	            #tempMoveBlkVariantRetVal := MOVE_BLK_VARIANT(SRC := #In_EventStatus.sts_Events,
	                                                                 COUNT := INT_TO_UDINT(#In_EventStatus.sts_NumEvents),
	                                                                 SRC_INDEX := 0,
	                                                                 DEST_INDEX := 0,
	                                                                 DEST => #Sts_EventSummation.sts_Events);
	            #Sts_EventSummation.sts_NumEvents := #In_EventStatus.sts_NumEvents;
	        ELSE
	            
	            #tempMoveBlkVariantRetVal := MOVE_BLK_VARIANT(SRC := #In_EventStatus.sts_Events,
	                                                                 COUNT := INT_TO_UDINT (#Sts_EventSummation.wrk_EventArraySize),
	                                                                 SRC_INDEX := 0,
	                                                                 DEST_INDEX := 0,
	                                                                 DEST => #Sts_EventSummation.sts_Events);
	            #Sts_EventSummation.sts_NumEvents := #Sts_EventSummation.wrk_EventArraySize;
	            #Sts_ErrorCode := 1;
	        END_IF;
	    
	   
	    END_IF;    
	END_IF;
	
	// update the output
	#Sts_NumEvents := #Sts_EventSummation.sts_NumEvents;
	
	// Set Category Bits
	#Sts_EventSummation.wrk_Category_0_Latched := (#Sts_EventSummation.wrk_Category_0_Latched OR #In_EventStatus.sts_Category_0_Latched);
	#Sts_EventSummation.wrk_Category_1_Latched := (#Sts_EventSummation.wrk_Category_1_Latched OR #In_EventStatus.sts_Category_1_Latched);
	#Sts_EventSummation.wrk_Category_2_Latched := (#Sts_EventSummation.wrk_Category_2_Latched OR #In_EventStatus.sts_Category_2_Latched);
	#Sts_EventSummation.wrk_Category_3_Latched := (#Sts_EventSummation.wrk_Category_3_Latched OR #In_EventStatus.sts_Category_3_Latched);
	#Sts_EventSummation.wrk_Category_4_Latched := (#Sts_EventSummation.wrk_Category_4_Latched OR #In_EventStatus.sts_Category_4_Latched);
	#Sts_EventSummation.wrk_Category_5_Latched := (#Sts_EventSummation.wrk_Category_5_Latched OR #In_EventStatus.sts_Category_5_Latched);
	#Sts_EventSummation.wrk_Category_6_Latched := (#Sts_EventSummation.wrk_Category_6_Latched OR #In_EventStatus.sts_Category_6_Latched);
	#Sts_EventSummation.wrk_Category_7_Latched := (#Sts_EventSummation.wrk_Category_7_Latched OR #In_EventStatus.sts_Category_7_Latched);
	#Sts_EventSummation.wrk_Category_8_Latched := (#Sts_EventSummation.wrk_Category_8_Latched OR #In_EventStatus.sts_Category_8_Latched);
	#Sts_EventSummation.wrk_Category_9_Latched := (#Sts_EventSummation.wrk_Category_9_Latched OR #In_EventStatus.sts_Category_9_Latched);
	
	#Sts_Category_0_Latched := #In_EventStatus.sts_Category_0_Latched;
	#Sts_Category_1_Latched := #In_EventStatus.sts_Category_1_Latched;
	#Sts_Category_2_Latched := #In_EventStatus.sts_Category_2_Latched;
	#Sts_Category_3_Latched := #In_EventStatus.sts_Category_3_Latched;
	#Sts_Category_4_Latched := #In_EventStatus.sts_Category_4_Latched;
	#Sts_Category_5_Latched := #In_EventStatus.sts_Category_5_Latched;
	#Sts_Category_6_Latched := #In_EventStatus.sts_Category_6_Latched;
	#Sts_Category_7_Latched := #In_EventStatus.sts_Category_7_Latched;
	#Sts_Category_8_Latched := #In_EventStatus.sts_Category_8_Latched;
	#Sts_Category_9_Latched := #In_EventStatus.sts_Category_9_Latched;
	
	#Sts_EventSummation.wrk_Category_0_NotLatched := #Sts_EventSummation.wrk_Category_0_NotLatched OR #In_EventStatus.sts_Category_0_NotLatched;
	#Sts_EventSummation.wrk_Category_1_NotLatched := #Sts_EventSummation.wrk_Category_1_NotLatched OR #In_EventStatus.sts_Category_1_NotLatched;
	#Sts_EventSummation.wrk_Category_2_NotLatched := #Sts_EventSummation.wrk_Category_2_NotLatched OR #In_EventStatus.sts_Category_2_NotLatched;
	#Sts_EventSummation.wrk_Category_3_NotLatched := #Sts_EventSummation.wrk_Category_3_NotLatched OR #In_EventStatus.sts_Category_3_NotLatched;
	#Sts_EventSummation.wrk_Category_4_NotLatched := #Sts_EventSummation.wrk_Category_4_NotLatched OR #In_EventStatus.sts_Category_4_NotLatched;
	#Sts_EventSummation.wrk_Category_5_NotLatched := #Sts_EventSummation.wrk_Category_5_NotLatched OR #In_EventStatus.sts_Category_5_NotLatched;
	#Sts_EventSummation.wrk_Category_6_NotLatched := #Sts_EventSummation.wrk_Category_6_NotLatched OR #In_EventStatus.sts_Category_6_NotLatched;
	#Sts_EventSummation.wrk_Category_7_NotLatched := #Sts_EventSummation.wrk_Category_7_NotLatched OR #In_EventStatus.sts_Category_7_NotLatched;
	#Sts_EventSummation.wrk_Category_8_NotLatched := #Sts_EventSummation.wrk_Category_8_NotLatched OR #In_EventStatus.sts_Category_8_NotLatched;
	#Sts_EventSummation.wrk_Category_9_NotLatched := #Sts_EventSummation.wrk_Category_9_NotLatched OR #In_EventStatus.sts_Category_9_NotLatched;
	
	#Sts_Category_0_NotLatched := #In_EventStatus.sts_Category_0_NotLatched;
	#Sts_Category_1_NotLatched := #In_EventStatus.sts_Category_1_NotLatched;
	#Sts_Category_2_NotLatched := #In_EventStatus.sts_Category_2_NotLatched;
	#Sts_Category_3_NotLatched := #In_EventStatus.sts_Category_3_NotLatched;
	#Sts_Category_4_NotLatched := #In_EventStatus.sts_Category_4_NotLatched;
	#Sts_Category_5_NotLatched := #In_EventStatus.sts_Category_5_NotLatched;
	#Sts_Category_6_NotLatched := #In_EventStatus.sts_Category_6_NotLatched;
	#Sts_Category_7_NotLatched := #In_EventStatus.sts_Category_7_NotLatched;
	#Sts_Category_8_NotLatched := #In_EventStatus.sts_Category_8_NotLatched;
	#Sts_Category_9_NotLatched := #In_EventStatus.sts_Category_9_NotLatched;
	
	#Sts_EventSummation.wrk_CurrentActiveEvent := #Sts_EventSummation.wrk_CurrentActiveEvent OR #In_EventStatus.sts_CurrentActiveEvent;
	
	#Sts_CurrentActiveEvent := #In_EventStatus.sts_CurrentActiveEvent;
	
	// Set Error Bit
	#Sts_Error := (#Sts_ErrorCode <> 0);
	
	//  -------------- END OF LOGIC -------------------------
	ENO := TRUE;   // Set the ENO output
	 
	
END_FUNCTION_BLOCK

FUNCTION_BLOCK "CPG_EventSummationEnd"
TITLE = CPG_EventSummationEnd
{ S7_Optimized_Access := 'TRUE' }
AUTHOR : 'tech.team.motioncontrol@siemens.com'
FAMILY : CPG
VERSION : 1.0
//Support: tech.team.motioncontrol@siemens.com
   VAR_IN_OUT 
      Sts_EventSummation : "CPG_typeEventSummation";   // Working event list data section
   END_VAR

   VAR 
      statFirstScan { ExternalAccessible := 'False'; ExternalVisible := 'False'; ExternalWritable := 'False'} : Bool;   // 0=1st scan of FB; set to 1 after 1st FB scan...
      statIndex { ExternalAccessible := 'False'; ExternalVisible := 'False'; ExternalWritable := 'False'} : Int;   // stat index
      statPrev_NumAllEvents { ExternalAccessible := 'False'; ExternalVisible := 'False'; ExternalWritable := 'False'} : Int;   // stat value needed with FOR loop
   END_VAR

   VAR_TEMP 
      tempZeroEvent : "CPG_typeEvent";   // null instance of UDT Event
   END_VAR


BEGIN
	//============================================================================================================
	// SIEMENS AG
	// (c)Copyright 2018 All Rights Reserved
	//------------------------------------------------------------------------------------------------------------
	// Project: CPG Template
	// Tested with: S7-1500 with FW version V2.1
	// Engineering: TIA Portal V14
	// Restrictions: ---
	// Requirements: S7-1500
	// Functionality:  Summarizes the "Data" from the equipment modules (from FB_EventManager) AND will create one list OF events FOR the unit machine.
	//                 It summarizes the data by finding the unit machine first out event and summarizes which category of events are active.
	//                 CPG_EventSummationBegin initializes the summation, and CPG_EventSummationEnd finalizes the summation.
	// Support: tech.team.motioncontrol@siemens.com
	//------------------------------------------------------------------------------------------------------------
	// Change log table:
	// Version       Date               Expert in charge    Changes applied
	//  01.00.00     01.01.2018         MP                  Initial Release & PackML V2.1  Renamed CPG V1.0
	//  01.01.00     29.05.2018         JP                  Adopted to styleguide
	//  01.00.01     13.06.2019         ThH                 Corrected handling of Bit 5; new Version CPG Template V1.0.1
	//============================================================================================================
	// Function Block : CPG_EventSummationEnd
	//============================================================================================================
	
	// ===========================================================================
	//  Begin the LOGIC section:
	// first scan logic
	IF #statFirstScan = FALSE THEN
	    // initialize & determine max array size
	    "CPG_ArrayLength"(arrayToBeSized := #Sts_EventSummation.sts_Events,
	                      arraySize => #Sts_EventSummation.wrk_EventArraySize);
	    
	    #statPrev_NumAllEvents := #Sts_EventSummation.wrk_EventArraySize;
	    
	    #statFirstScan := TRUE;            // set the first scan bit
	END_IF;
	
	// Cleanup the summation - This FB is to be called after the numerous "FB_PMLe_EventSum" calls.
	IF #statPrev_NumAllEvents > #Sts_EventSummation.sts_NumEvents THEN
	    
	    FOR #statIndex := #Sts_EventSummation.sts_NumEvents TO (#statPrev_NumAllEvents-1) DO
	        #Sts_EventSummation.sts_Events[#statIndex]:= #tempZeroEvent;   // clear event area of cleared alarms
	    END_FOR;
	    
	END_IF;
	    
	#statPrev_NumAllEvents := #Sts_EventSummation.sts_NumEvents;     
	
	// Update the output bits from work area
	#Sts_EventSummation.sts_Category_0_Latched := #Sts_EventSummation.wrk_Category_0_Latched;
	#Sts_EventSummation.sts_Category_1_Latched := #Sts_EventSummation.wrk_Category_1_Latched;
	#Sts_EventSummation.sts_Category_2_Latched := #Sts_EventSummation.wrk_Category_2_Latched;
	#Sts_EventSummation.sts_Category_3_Latched := #Sts_EventSummation.wrk_Category_3_Latched;
	#Sts_EventSummation.sts_Category_4_Latched := #Sts_EventSummation.wrk_Category_4_Latched;
	#Sts_EventSummation.sts_Category_5_Latched := #Sts_EventSummation.wrk_Category_5_Latched;
	#Sts_EventSummation.sts_Category_6_Latched := #Sts_EventSummation.wrk_Category_6_Latched;
	#Sts_EventSummation.sts_Category_7_Latched := #Sts_EventSummation.wrk_Category_7_Latched;
	#Sts_EventSummation.sts_Category_8_Latched := #Sts_EventSummation.wrk_Category_8_Latched;
	#Sts_EventSummation.sts_Category_9_Latched := #Sts_EventSummation.wrk_Category_9_Latched;
	
	#Sts_EventSummation.sts_Category_0_NotLatched := #Sts_EventSummation.wrk_Category_0_NotLatched;
	#Sts_EventSummation.sts_Category_1_NotLatched := #Sts_EventSummation.wrk_Category_1_NotLatched;
	#Sts_EventSummation.sts_Category_2_NotLatched := #Sts_EventSummation.wrk_Category_2_NotLatched;
	#Sts_EventSummation.sts_Category_3_NotLatched := #Sts_EventSummation.wrk_Category_3_NotLatched;
	#Sts_EventSummation.sts_Category_4_NotLatched := #Sts_EventSummation.wrk_Category_4_NotLatched;
	#Sts_EventSummation.sts_Category_5_NotLatched := #Sts_EventSummation.wrk_Category_5_NotLatched;
	#Sts_EventSummation.sts_Category_6_NotLatched := #Sts_EventSummation.wrk_Category_6_NotLatched;
	#Sts_EventSummation.sts_Category_7_NotLatched := #Sts_EventSummation.wrk_Category_7_NotLatched;
	#Sts_EventSummation.sts_Category_8_NotLatched := #Sts_EventSummation.wrk_Category_8_NotLatched;
	#Sts_EventSummation.sts_Category_9_NotLatched := #Sts_EventSummation.wrk_Category_9_NotLatched;
	
	#Sts_EventSummation.sts_CurrentActiveEvent  := #Sts_EventSummation.wrk_CurrentActiveEvent; 
	    
	//  -------------- END OF LOGIC -------------------------
	ENO := TRUE;   // Set the ENO output
	
END_FUNCTION_BLOCK

FUNCTION_BLOCK "CPG_AlarmMove"
TITLE = CPG_AlarmMove
{ S7_Optimized_Access := 'TRUE' }
AUTHOR : 'tech.team.motioncontrol@siemens.com'
FAMILY : CPG
VERSION : 1.0
//Support: tech.team.motioncontrol@siemens.com
   VAR_INPUT 
      Sts_NumEvents { ExternalAccessible := 'False'; ExternalVisible := 'False'; ExternalWritable := 'False'} : Int;   // Number of Active Alarms
   END_VAR

   VAR_OUTPUT 
      Sts_Error { ExternalAccessible := 'False'; ExternalVisible := 'False'; ExternalWritable := 'False'} : Bool;   // Error Status.  0=no error, 1=error
      Sts_ErrorCode { ExternalAccessible := 'False'; ExternalVisible := 'False'; ExternalWritable := 'False'} : Int;   // Error code / number
   END_VAR

   VAR_IN_OUT 
      source : Array[0.."CPG_NO_OF_STS_ELEMENTS_EVENT_SUM_UPPER_LIM"] of "CPG_typeEvent";   // source location of the machine alarms
      destination : Array[0.."CPG_NO_OF_ADMIN_EVENTS_UPPER_LIM"] of "CPG_typeEvent";   // destination location of the PackTag alarms
   END_VAR

   VAR 
      statSourceNumEvents { ExternalAccessible := 'False'; ExternalVisible := 'False'; ExternalWritable := 'False'} : Int;   // MAX # OF Events - source event list
      statDestinationNumEvents { ExternalAccessible := 'False'; ExternalVisible := 'False'; ExternalWritable := 'False'} : Int;   // MAX # OF Events - destination event list
      statIndex { ExternalAccessible := 'False'; ExternalVisible := 'False'; ExternalWritable := 'False'} : Int;   // index value
      statPrevNumEvents { ExternalAccessible := 'False'; ExternalVisible := 'False'; ExternalWritable := 'False'} : Int;   // previous number of events
      statZeroEvent { ExternalAccessible := 'False'; ExternalVisible := 'False'; ExternalWritable := 'False'} : "CPG_typeEvent";   // blank event
      statWrkNumEvents { ExternalAccessible := 'False'; ExternalVisible := 'False'; ExternalWritable := 'False'} : Int;   // working number of active events
   END_VAR


BEGIN
	//============================================================================================================
	// SIEMENS AG
	// (c)Copyright 2018 All Rights Reserved
	//------------------------------------------------------------------------------------------------------------
	// Project: CPG Template
	// Tested with: S7-1500 with FW version V2.1
	// Engineering: TIA Portal V14
	// Restrictions: ---
	// Requirements: S7-1500
	// Functionality: move alarm structures 
	// Support: tech.team.motioncontrol@siemens.com
	//------------------------------------------------------------------------------------------------------------
	// Change log table:
	// Version       Date               Expert in charge    Changes applied
	//  01.00.00     01.01.2018         MP                  Initial Release & PackML V1.5  Renamed CPG V1.0
	//  01.01.00     22.05.2018         JP                  Adopted to styleguide
	//============================================================================================================
	// Function : CPG_AlarmMove
	//============================================================================================================
	
	
	// initialize & determine max array size
	"CPG_ArrayLength"(arrayToBeSized := #source,
	                  arraySize => #statSourceNumEvents);
	
	"CPG_ArrayLength"(arrayToBeSized := #destination,
	                  arraySize => #statDestinationNumEvents);
	
	#statWrkNumEvents := #Sts_NumEvents;
	
	IF (#statDestinationNumEvents < #statSourceNumEvents) AND (#statDestinationNumEvents < #Sts_NumEvents) THEN
	  #statWrkNumEvents := #statDestinationNumEvents;
	END_IF;
	
	IF (#statSourceNumEvents < #statDestinationNumEvents) AND (#statSourceNumEvents < #Sts_NumEvents) THEN
	  #statWrkNumEvents := #statSourceNumEvents;
	END_IF;
	
	FOR #statIndex := 0 TO #statWrkNumEvents - 1 DO
	  #destination[#statIndex] := #source[#statIndex];
	END_FOR;
	
	// Clean up event list
	IF #statPrevNumEvents > #statWrkNumEvents THEN
	  FOR #statIndex := #statWrkNumEvents TO #statPrevNumEvents - 1 DO
	    #destination[#statIndex] := #statZeroEvent;
	  END_FOR;
	END_IF;
	
	#statPrevNumEvents := #statWrkNumEvents;
	
	//  -------------- END OF LOGIC -------------------------
	ENO := TRUE;   // Set the ENO output
END_FUNCTION_BLOCK

FUNCTION_BLOCK "CPG_AlarmHistory"
TITLE = CPG_AlarmHistory
{ S7_Optimized_Access := 'TRUE' }
AUTHOR : 'tech.team.motioncontrol@siemens.com'
FAMILY : CPG
VERSION : 1.1
//Support: tech.team.motioncontrol@siemens.com
   VAR_OUTPUT 
      alarmHistoryArraySize : Int;   // Size of Alarm History - number of alarm array elements
   END_VAR

   VAR_IN_OUT 
      inStopReasonAlarm : "CPG_typeEvent";   // Input - Stop Reason Alarm (structure)
      stsAlarmHistory : Array[0.."CPG_NO_OF_ADMIN_EVENTS_HISTORY_UPPER_LIM"] of "CPG_typeEvent";   // Status- Alarm History Log
   END_VAR

   VAR 
      statAlarmArraySize { ExternalAccessible := 'False'; ExternalVisible := 'False'; ExternalWritable := 'False'} : Int;   // Max # of Events in the Alarm History Array
      statTriggerOsPos { ExternalAccessible := 'False'; ExternalVisible := 'False'; ExternalWritable := 'False'} : Bool;   // Trigger One Shot - positive edge
      statTriggerOsNeg { ExternalAccessible := 'False'; ExternalVisible := 'False'; ExternalWritable := 'False'} : Bool;   // Trigger One Shot - negative edge
      statErrorRtc { ExternalAccessible := 'False'; ExternalVisible := 'False'; ExternalWritable := 'False'} : Int;   // Error code for reading of Real Time Clock
      statEventCurDateTime {InstructionName := 'DTL'; LibVersion := '1.0'; ExternalAccessible := 'False'; ExternalVisible := 'False'; ExternalWritable := 'False'} : DTL;   // temp value for current date & time
      statFirstScan { ExternalAccessible := 'False'; ExternalVisible := 'False'; ExternalWritable := 'False'} : Bool;   // 0=1st scan of FB; set to 1 after 1st FB scan...
   END_VAR

   VAR_TEMP 
      tempIndex : Int;   // temp index value
   END_VAR

   VAR CONSTANT 
      ZERO : Int := 0;   // constant = 0
      NEGATIVE_ONE : Int := -1;   // constant = -1
   END_VAR


BEGIN
	//============================================================================================================
	// SIEMENS AG
	// (c)Copyright 2018 All Rights Reserved
	//------------------------------------------------------------------------------------------------------------
	// Project: CPG Template
	// Tested with: S7-1500 with FW version V2.1
	// Engineering: TIA Portal V14
	// Restrictions: ---
	// Requirements: S7-1500
	// Functionality: used to capture the current Stop ReasonAlarm (i.e. 'Machine)
	//                First Fault to the "PackTags" AlarmHistory log.
	// Support: tech.team.motioncontrol@siemens.com
	//------------------------------------------------------------------------------------------------------------
	// Change log table:
	// Version       Date               Expert in charge    Changes applied
	//  01.00.00     01.01.2018         MP                  Initial Release & PackML V1.5  Renamed CPG V1.0
	//  01.01.00     22.05.2018         JP                  Adopted to styleguide
	//  01.01.01     01.05.2020         KB                  Changed RD_SYS_T -> RD_LOC_T
	//============================================================================================================
	// Function : CPG_AlarmHistory
	//============================================================================================================
	
	// First Scan Logic
	IF #statFirstScan = FALSE THEN
	  "CPG_ArrayLength"(arrayToBeSized := #stsAlarmHistory,
	                    arraySize => #statAlarmArraySize);
	
	  // Update number of array elements in Alarm History Array (used for Admin.AlarmHistoryExtent)
	  #alarmHistoryArraySize := #statAlarmArraySize;
	
	  #statFirstScan := TRUE;      // Set the FB 1st Scan Bit
	END_IF;
	
	// Positive Trigger
	IF #inStopReasonAlarm.Trigger = TRUE AND #statTriggerOsPos = FALSE THEN
	  // execute code for new incoming event
	  #statTriggerOsPos := TRUE;   // Set the One Shot Bit 
	
	  // Index the existing Alarm History Array (FIFO).
	  FOR #tempIndex := #statAlarmArraySize - 1 TO 1 BY -1 DO
	    #stsAlarmHistory[#tempIndex] := #stsAlarmHistory[#tempIndex - 1];
	  END_FOR;
	
	  // Update the Array[0] with the current alarm information
	  #stsAlarmHistory[0] := #inStopReasonAlarm;
	END_IF;
	
	IF #inStopReasonAlarm.Trigger = FALSE AND #statTriggerOsPos = TRUE THEN
	  // Reset the One Shot Bit
	  #statTriggerOsPos := FALSE;  // Reset the One Shot Bit
	END_IF;
	
	// Negative Trigger
	IF #inStopReasonAlarm.Trigger = FALSE AND #statTriggerOsNeg = FALSE THEN
	  // Execute code for new incoming event
	  #statTriggerOsNeg := TRUE;    // Set the One Shot Bit
	  // Capture the Alarm Ack. Time
	  #statErrorRtc := RD_LOC_T(#statEventCurDateTime);     // Read the Real Time Clock
	  #stsAlarmHistory[0].AckDateTimeDTL := #statEventCurDateTime; // Update acknowledge time
	END_IF;
	
	IF #inStopReasonAlarm.Trigger = TRUE AND #statTriggerOsPos = TRUE THEN
	  // Reset the One Shot Bit
	  #statTriggerOsNeg := FALSE;   // Reset the One Shot Bit
	END_IF;
	
	//  -------------- END OF LOGIC -------------------------
	ENO := TRUE;   // Set the ENO output
END_FUNCTION_BLOCK

FUNCTION_BLOCK "CPG_EventSortFilter"
TITLE = CPG_EventSortFilter
{ S7_Optimized_Access := 'TRUE' }
AUTHOR : 'tech.team.motioncontrol@siemens.com'
FAMILY : CPG
VERSION : 1.0
//Support: tech.team.motioncontrol@siemens.com
   VAR_INPUT 
      Cfg_EventListOffset { ExternalAccessible := 'False'; ExternalVisible := 'False'; ExternalWritable := 'False'} : Int;   // Commanded event list offset (used for scrolling)
      Cfg_FilterCategory { ExternalAccessible := 'False'; ExternalVisible := 'False'; ExternalWritable := 'False'} : Int;   // Filtered category number
      Cfg_TimeSortDirection { ExternalAccessible := 'False'; ExternalVisible := 'False'; ExternalWritable := 'False'} : Bool;   // 1=newest first; 0=oldest first
      Cmd_FilterActiveEvents { ExternalAccessible := 'False'; ExternalVisible := 'False'; ExternalWritable := 'False'} : Bool;   // 1=only show active events; 0=show all events
      Cmd_FilterCategory { ExternalAccessible := 'False'; ExternalVisible := 'False'; ExternalWritable := 'False'} : Bool;   // Filter events to show only selected category number
      Cmd_SortCategory { ExternalAccessible := 'False'; ExternalVisible := 'False'; ExternalWritable := 'False'} : Bool;   // 1=Sort events by ascending category number
   END_VAR

   VAR_OUTPUT 
      Sts_EventListOffset { ExternalAccessible := 'False'; ExternalVisible := 'False'; ExternalWritable := 'False'} : Int;   // Actual event list offset
      Sts_FilterExcludedNumEvents { ExternalAccessible := 'False'; ExternalVisible := 'False'; ExternalWritable := 'False'} : Int;   // The number of events excluded by filtering
      Sts_SortFilterNumEvents { ExternalAccessible := 'False'; ExternalVisible := 'False'; ExternalWritable := 'False'} : Int;   // Number of events in the sorted or filtered event list
   END_VAR

   VAR_IN_OUT 
      In_Events : Array[0.."CPG_NO_OF_STS_ELEMENTS_EVENT_SUM_UPPER_LIM"] of "CPG_typeEvent";   // Input Event list to be sorted and/or filtered
      In_NumEvents { ExternalAccessible := 'False'; ExternalVisible := 'False'; ExternalWritable := 'False'} : Int;   // Number of events to be sorted and/or filtered
      Sts_SortFilterEventList : Array[0.."CPG_NO_OF_HMI_SORT_EVENTS_UPPER_LIM"] of "CPG_typeEvent";   // Output sorted and/or filtered event list
   END_VAR

   VAR 
      statFirstScan { ExternalAccessible := 'False'; ExternalVisible := 'False'; ExternalWritable := 'False'} : Bool;   // stat first scan bit
      statCatIndex { ExternalAccessible := 'False'; ExternalVisible := 'False'; ExternalWritable := 'False'} : Int;   // stat category index
      statCopiedIndex { ExternalAccessible := 'False'; ExternalVisible := 'False'; ExternalWritable := 'False'} : Int;   // stat copied index
      statFilterActive { ExternalAccessible := 'False'; ExternalVisible := 'False'; ExternalWritable := 'False'} : Bool;   // stat filter active = 1
      statFilterCategory { ExternalAccessible := 'False'; ExternalVisible := 'False'; ExternalWritable := 'False'} : Bool;   // stat filter category
      statFilteredIndex { ExternalAccessible := 'False'; ExternalVisible := 'False'; ExternalWritable := 'False'} : Int;   // stat filtered index
      statIndex { ExternalAccessible := 'False'; ExternalVisible := 'False'; ExternalWritable := 'False'} : Int;   // stat index
      statLocalEventOffset { ExternalAccessible := 'False'; ExternalVisible := 'False'; ExternalWritable := 'False'} : Int;   // stat local event offset
      statMaxInputSize { ExternalAccessible := 'False'; ExternalVisible := 'False'; ExternalWritable := 'False'} : Int;   // stat max input size
      statMaxLocalInputSize { ExternalAccessible := 'False'; ExternalVisible := 'False'; ExternalWritable := 'False'} : Int;   // stat max  local input size
      statMaxOutputSize { ExternalAccessible := 'False'; ExternalVisible := 'False'; ExternalWritable := 'False'} : Int;   // stat max output size
      statMaxParameterInputSize { ExternalAccessible := 'False'; ExternalVisible := 'False'; ExternalWritable := 'False'} : Int;   // stat max parameter input size
      statNumDisplayedEvents { ExternalAccessible := 'False'; ExternalVisible := 'False'; ExternalWritable := 'False'} : Int;   // stat num displayed events
      statNumFilteredEvents { ExternalAccessible := 'False'; ExternalVisible := 'False'; ExternalWritable := 'False'} : Int;   // stat num of filtered events
      statPrevNumEvents { ExternalAccessible := 'False'; ExternalVisible := 'False'; ExternalWritable := 'False'} : Int;   // stat previous number of events
      statSortedIndex { ExternalAccessible := 'False'; ExternalVisible := 'False'; ExternalWritable := 'False'} : Int;   // stat sorted index
      statFilteredEventList { ExternalAccessible := 'False'; ExternalVisible := 'False'; ExternalWritable := 'False'} : Array[0.."CPG_NO_OF_STS_ELEMENTS_EVENT_SUM_UPPER_LIM"] of "CPG_typeEvent";   // stat sorted event list
      statZeroEvent { ExternalAccessible := 'False'; ExternalVisible := 'False'; ExternalWritable := 'False'} : "CPG_typeEvent";   // stat zeroized event list
   END_VAR

   VAR_TEMP 
      tempMoveBlkVariantRetVal : Int;   // temp return value for BlockMoveVariant
   END_VAR

   VAR CONSTANT 
      ZERO_VALUE : Int := 0;
   END_VAR


BEGIN
	//============================================================================================================
	// SIEMENS AG
	// (c)Copyright 2018 All Rights Reserved
	//------------------------------------------------------------------------------------------------------------
	// Project: CPG Template
	// Tested with: S7-1500 with FW version V2.1
	// Engineering: TIA Portal V14
	// Restrictions: ---
	// Requirements: S7-1500
	// Functionality: Control Event Sort Filter commands
	// Support: tech.team.motioncontrol@siemens.com
	//------------------------------------------------------------------------------------------------------------
	// Change log table:
	// Version       Date               Expert in charge    Changes applied
	//  01.00.00     01.01.2018         MP                  Initial Release & PackML V2.1  Renamed CPG V1.0
	//  01.01.00     29.05.2018         JP                  Adopted to styleguide
	//============================================================================================================
	// Function : CPG_EventSortFilter
	//============================================================================================================
	
	IF #statFirstScan = FALSE THEN
	    // initialize & determine max array size
	    // input array size (i.e. Array[0.."CPG_NO_STS_ELEMENTS_EVENT_STATUS"] of "typeCPG_Event")
	    "CPG_ArrayLength"(arrayToBeSized := #In_Events,
	                      arraySize => #statMaxParameterInputSize);
	    
	    //output array size for HMI (i.e. Array[0.."CPG_NO_HMI_SORT_EVENTS"] of "typeCPG_Event")
	    "CPG_ArrayLength"(arrayToBeSized := #Sts_SortFilterEventList,
	                      arraySize => #statMaxOutputSize);
	    
	    // internal/temporary array size (i.e. Array[0.."CPG_NO_STS_ELEMENTS_EVENT_STATUS"] of "typeCPG_Event")   
	    "CPG_ArrayLength"(arrayToBeSized := #statFilteredEventList,
	                              arraySize => #statMaxLocalInputSize);
	    
	    //Take smallest aray as the maximum number of input events to filter and sort
	    IF #statMaxParameterInputSize > #statMaxLocalInputSize THEN
	        #statMaxInputSize := #statMaxLocalInputSize;
	    ELSE
	        #statMaxInputSize := #statMaxParameterInputSize;
	    END_IF;
	    // clear the output sort buffer
	    FOR #statIndex := 0 TO #statMaxOutputSize - 1 DO
	        #Sts_SortFilterEventList[#statIndex] := #statZeroEvent;
	    END_FOR;
	    
	    #statFirstScan := TRUE;            // set the first scan bit 
	END_IF;
	// End of First Scan Section
	
	
	// Main Filter Logic
	
	#statFilteredIndex := 0;
	// sort by ascending OR descending?
	IF #Cfg_TimeSortDirection THEN
	    #statIndex := #In_NumEvents - 1;  // newest events first
	ELSE
	    #statIndex := 0;   // oldest events first
	END_IF;
	
	IF #In_NumEvents > 0 THEN
	    
	    REPEAT
	        #statFilterCategory := 0;
	        #statFilterActive := 0;
	        IF #Cmd_FilterCategory AND (#In_Events[#statIndex].Category = #Cfg_FilterCategory) THEN
	            #statFilterCategory := 1;
	        END_IF;
	        IF #Cmd_FilterActiveEvents AND (#In_Events[#statIndex].Trigger) THEN
	            #statFilterActive := 1;
	        END_IF;
	        
	        IF ((#Cmd_FilterCategory AND #statFilterCategory) OR NOT (#Cmd_FilterCategory)) AND ((#Cmd_FilterActiveEvents AND #statFilterActive) OR NOT (#Cmd_FilterActiveEvents)) THEN
	            #statFilteredEventList[#statFilteredIndex] := #In_Events[#statIndex];
	            #statFilteredIndex := #statFilteredIndex + 1;
	        END_IF;
	        
	        IF #Cfg_TimeSortDirection THEN
	            #statIndex := #statIndex - 1;
	        ELSE
	            #statIndex := #statIndex + 1;
	        END_IF;
	        
	    UNTIL #statFilteredIndex >= #In_NumEvents OR #statFilteredIndex >= #statMaxInputSize OR #statIndex < 0 OR #statIndex >= #In_NumEvents END_REPEAT;
	END_IF;
	
	#statNumFilteredEvents := #statFilteredIndex;
	
	#Sts_SortFilterNumEvents := #statNumFilteredEvents;
	#Sts_FilterExcludedNumEvents := #In_NumEvents - #statNumFilteredEvents;
	
	//Sanitize and limit Cfg_EventListOffset, offset cannot go past the last event
	IF #Cfg_EventListOffset > #statNumFilteredEvents - 1 THEN
	    #statLocalEventOffset := #statNumFilteredEvents - 1;
	ELSE
	    #statLocalEventOffset := #Cfg_EventListOffset;
	END_IF;
	
	IF #statLocalEventOffset < 0 THEN
	    #statLocalEventOffset := 0;
	END_IF;
	#Sts_EventListOffset := #statLocalEventOffset;
	
	#statSortedIndex := 0;
	#statCopiedIndex := 0;
	
	//Category sorting loops
	IF #Cmd_SortCategory THEN
	    IF #statNumFilteredEvents <> 0 THEN
	        #statCatIndex := 0;
	        REPEAT //Repeat for categories 0-9
	            #statIndex := 0;
	            
	            REPEAT //Repeat for every event in the filtered list
	                //If the category matches, add to the list
	                
	                IF #statCatIndex = #statFilteredEventList[#statIndex].Category THEN
	                    //Track sorted index separate from copied index.  
	                    //This allows a "hypothetical" sort when an offset is applied, without using memory for a non-offset sorted list
	                    IF (#statSortedIndex >= #statLocalEventOffset) THEN
	                        #Sts_SortFilterEventList[#statCopiedIndex] := #statFilteredEventList[#statIndex];
	                        #statCopiedIndex := #statCopiedIndex + 1;
	                    END_IF;
	                    #statSortedIndex := #statSortedIndex + 1;
	                END_IF;
	                
	                IF #statCopiedIndex >= #statMaxOutputSize THEN
	                    EXIT; //EXIT unsorted loop
	                END_IF;
	                
	                #statIndex := #statIndex + 1;
	            UNTIL #statIndex >= #statNumFilteredEvents END_REPEAT;
	            
	            IF #statCopiedIndex >= #statMaxOutputSize THEN
	                EXIT; //EXIT category loop
	            END_IF;
	            #statCatIndex := #statCatIndex + 1;
	        UNTIL #statCatIndex > 9 END_REPEAT;
	        
	        //Handle display of events in the case the category is not 0-9, but do not sort in order for scan time purposes
	        //Only for special cases
	        IF #statCopiedIndex < #statMaxOutputSize - 1 AND #statSortedIndex <> #statNumFilteredEvents THEN
	            #statIndex := 0;
	            REPEAT
	                IF #statFilteredEventList[#statIndex].Category > 9 THEN
	                    IF (#statSortedIndex >= #statLocalEventOffset) THEN
	                        #Sts_SortFilterEventList[#statCopiedIndex] := #statFilteredEventList[#statIndex];
	                        #statCopiedIndex := #statCopiedIndex + 1;
	                    END_IF;
	                    
	                    #statSortedIndex := #statSortedIndex + 1;
	                    
	                END_IF;
	                
	                
	                IF #statCopiedIndex >= #statMaxOutputSize THEN
	                    EXIT;
	                END_IF;
	                
	                #statIndex := #statIndex + 1;
	                
	            UNTIL #statIndex >= #statNumFilteredEvents END_REPEAT;
	            
	        END_IF;
	        
	    END_IF;
	    
	ELSE
	    //If no category sorting is done, copy the entire filtered list and apply any offset
	    #statCopiedIndex := #statNumFilteredEvents - #statLocalEventOffset;
	    
	    IF #statCopiedIndex > #statMaxOutputSize THEN
	        #statCopiedIndex := #statMaxOutputSize;
	    ELSIF #statCopiedIndex < 0 THEN
	        #statCopiedIndex := 0;
	    END_IF;
	    
	    #tempMoveBlkVariantRetVal := MOVE_BLK_VARIANT(SRC := #statFilteredEventList, COUNT := DINT_TO_UDINT(#statCopiedIndex), SRC_INDEX := #statLocalEventOffset, DEST_INDEX := #ZERO_VALUE, DEST => #Sts_SortFilterEventList);
	    
	END_IF;
	
	#statNumDisplayedEvents := #statCopiedIndex;
	
	// Clean up event list
	IF #statPrevNumEvents > #statNumDisplayedEvents THEN
	    FOR #statIndex := #statNumDisplayedEvents TO #statPrevNumEvents - 1 DO
	        #Sts_SortFilterEventList[#statIndex] := #statZeroEvent;
	    END_FOR;
	END_IF;
	
	#statPrevNumEvents := #statNumDisplayedEvents;
	
	//  -------------- END OF LOGIC -------------------------
	ENO := TRUE;   // Set the ENO output
END_FUNCTION_BLOCK

FUNCTION_BLOCK "CPG_MsgScroll"
TITLE = CPG_Msg_Scroll
{ S7_Optimized_Access := 'TRUE' }
AUTHOR : 'tech.team.motioncontrol@siemens.com'
FAMILY : CPG
VERSION : 1.0
//Support: tech.team.motioncontrol@siemens.com
   VAR_INPUT 
      Trigger { ExternalAccessible := 'False'; ExternalVisible := 'False'; ExternalWritable := 'False'} : Bool;   // input trigger to enable scroll logic
      NumEvents { ExternalAccessible := 'False'; ExternalVisible := 'False'; ExternalWritable := 'False'} : Int;   // input value with number of active events
      In_Events { ExternalAccessible := 'False'; ExternalVisible := 'False'; ExternalWritable := 'False'} : Array[0.."CPG_NO_OF_HMI_SORT_EVENTS_UPPER_LIM"] of "CPG_typeEvent";   // incoming events list
   END_VAR

   VAR_OUTPUT 
      Msg_Scroll { ExternalAccessible := 'False'; ExternalVisible := 'False'; ExternalWritable := 'False'} : String[40];   // message output value
   END_VAR

   VAR 
      statScrollIndex { ExternalAccessible := 'False'; ExternalVisible := 'False'; ExternalWritable := 'False'} : Int;   // index value for scroll logic
      statTriggerOS { ExternalAccessible := 'False'; ExternalVisible := 'False'; ExternalWritable := 'False'} : Bool;   // one shot trigger
      statMaxSize { ExternalAccessible := 'False'; ExternalVisible := 'False'; ExternalWritable := 'False'} : Int;   // max size
   END_VAR

   VAR_TEMP 
      tempScroll_Index_Max : Int;   // max value for scroll index
   END_VAR


BEGIN
	//============================================================================================================
	// SIEMENS AG
	// (c)Copyright 2018 All Rights Reserved
	//------------------------------------------------------------------------------------------------------------
	// Project: CPG Template
	// Tested with: S7-1500 with FW version V2.1
	// Engineering: TIA Portal V14
	// Restrictions: ---
	// Requirements: S7-1500
	// Functionality:  Used to scoll messages from an array of the active events to a single string for display on the HMI
	// Support: tech.team.motioncontrol@siemens.com
	//------------------------------------------------------------------------------------------------------------
	// Change log table:
	// Version       Date               Expert in charge    Changes applied
	//  01.00.00     01.01.2018         MP                  Initial Release & PackML V2.1  Renamed CPG V1.0
	//  01.01.00     29.05.2018         JP                  Adopted to styleguide
	//============================================================================================================
	// Function Block : CPG_Msg_Scroll
	//============================================================================================================
	
	
	
	// ===========================================================================
	//  Begin the LOGIC section:
	// initialize & determine max array size
	"CPG_ArrayLength"(arrayToBeSized := #In_Events,
	                         arraySize => #statMaxSize);
	
	IF #NumEvents > #statMaxSize THEN
	    #tempScroll_Index_Max := #statMaxSize;
	ELSE
	    #tempScroll_Index_Max := #NumEvents;
	END_IF;
	    
	// Statement Section 
	IF #Trigger AND NOT #statTriggerOS THEN
	    #statScrollIndex := #statScrollIndex + 1;  // increment the index
	    
	    IF  #statScrollIndex > #tempScroll_Index_Max - 1 THEN
	            #statScrollIndex := 0;
	        END_IF;
	        
	   #Msg_Scroll := #In_Events[#statScrollIndex].Message;      // move the message from the UDT_Event structure to string output.  
	
	    #statTriggerOS := TRUE;              // Set the trigger OS bit
	END_IF;
	
	IF NOT #Trigger AND #statTriggerOS THEN
	    #statTriggerOS := FALSE;
	END_IF;
	
	//  -------------- END OF LOGIC -------------------------
	ENO := TRUE;   // Set the ENO output
	
END_FUNCTION_BLOCK

FUNCTION_BLOCK "CPG_ParetoAnalysis"
TITLE = CPG_ParetoAnalysis
{ S7_Optimized_Access := 'TRUE' }
AUTHOR : 'tech.team.motioncontrol@siemens.com'
FAMILY : CPG
VERSION : 1.1
//Support: tech.team.motioncontrol@siemens.com
   VAR_INPUT 
      ID { ExternalAccessible := 'False'; ExternalVisible := 'False'; ExternalWritable := 'False'} : DInt;   // ID of the current alarm (0 if no alarm active)
      message { ExternalAccessible := 'False'; ExternalVisible := 'False'; ExternalWritable := 'False'} : String[40];   // Text of the current alarm
      resetPareto { ExternalAccessible := 'False'; ExternalVisible := 'False'; ExternalWritable := 'False'} : Bool;   // Rising edge resets statistics
      sort { ExternalAccessible := 'False'; ExternalVisible := 'False'; ExternalWritable := 'False'} : Int;   // Choose metric to sort by (0=totalDowntime, 1=percentOccurred, 2=timesOccurred, 3=MTTR)
   END_VAR

   VAR_OUTPUT 
      totalStops { ExternalAccessible := 'False'; ExternalVisible := 'False'; ExternalWritable := 'False'} : UInt;   // Total stops due to all faults
      totalTimeSinceReset { ExternalAccessible := 'False'; ExternalVisible := 'False'; ExternalWritable := 'False'} : Real;   // Total time in minutes since reset
      totalUptime { ExternalAccessible := 'False'; ExternalVisible := 'False'; ExternalWritable := 'False'} : Real;   // Total uptime in minutes
      totalDowntime { ExternalAccessible := 'False'; ExternalVisible := 'False'; ExternalWritable := 'False'} : Real;   // Total downtime in minutes
      percentUptime { ExternalAccessible := 'False'; ExternalVisible := 'False'; ExternalWritable := 'False'} : Real;   // Percent of total time since reset that was uptime
      MTTR { ExternalAccessible := 'False'; ExternalVisible := 'False'; ExternalWritable := 'False'} : Real;   // Mean time to return
      MTBF { ExternalAccessible := 'False'; ExternalVisible := 'False'; ExternalWritable := 'False'} : Real;   // Mean time between failures
   END_VAR

   VAR_IN_OUT 
      paretoData : Array[0.."CPG_PARTEO_NO_OF_ERRORS_UPPER_LIM"] of "CPG_typePareto";   // Alarm data structure
   END_VAR

   VAR 
      statFirstScan { ExternalAccessible := 'False'; ExternalVisible := 'False'; ExternalWritable := 'False'} : Bool := TRUE;   // Indicate first scan
      statStopReasonOld { ExternalAccessible := 'False'; ExternalVisible := 'False'; ExternalWritable := 'False'} : DInt;   // The last stop reason
      statResetParetoOld { ExternalAccessible := 'False'; ExternalVisible := 'False'; ExternalWritable := 'False'} : Bool;   // Reset on the rising edge of resetPareto
      statEntryFound { ExternalAccessible := 'False'; ExternalVisible := 'False'; ExternalWritable := 'False'} : Bool;   // Alarm code exists already
      statCurrentTimestamp {InstructionName := 'DTL'; LibVersion := '1.0'; ExternalAccessible := 'False'; ExternalVisible := 'False'; ExternalWritable := 'False'} : DTL;   // Current local time
      statPrevTimestamp {InstructionName := 'DTL'; LibVersion := '1.0'; ExternalAccessible := 'False'; ExternalVisible := 'False'; ExternalWritable := 'False'} : DTL;   // Previous local time stamp
      statResetTimestamp {InstructionName := 'DTL'; LibVersion := '1.0'; ExternalAccessible := 'False'; ExternalVisible := 'False'; ExternalWritable := 'False'} : DTL;   // Time when reset
      statSameCurrentTimestamp { ExternalAccessible := 'False'; ExternalVisible := 'False'; ExternalWritable := 'False'} : Date_And_Time;   // New current time when same alarm is present
      statBaseDowntime { ExternalAccessible := 'False'; ExternalVisible := 'False'; ExternalWritable := 'False'} : Real;   // Set time when alarm doesn't change
      statIndex { ExternalAccessible := 'False'; ExternalVisible := 'False'; ExternalWritable := 'False'} : Int;   // Current index in the alarm array
      statTotalStops { ExternalAccessible := 'False'; ExternalVisible := 'False'; ExternalWritable := 'False'} : UInt;   // Total number of alarm stops
      statTotalDowntime { ExternalAccessible := 'False'; ExternalVisible := 'False'; ExternalWritable := 'False'} : Real;   // Total machine downtime
      statOverallMTTR { ExternalAccessible := 'False'; ExternalVisible := 'False'; ExternalWritable := 'False'} : Real;   // Overall total downtime/ Total stops
      statPrevTotalUptime { ExternalAccessible := 'False'; ExternalVisible := 'False'; ExternalWritable := 'False'} : Real;   // Previous total uptime
      instShellSortPareto { ExternalAccessible := 'False'; ExternalVisible := 'False'; ExternalWritable := 'False'} : "CPG_ShellSortPareto";   // Sort alarm array
      statSort { ExternalAccessible := 'False'; ExternalVisible := 'False'; ExternalWritable := 'False'} : String[30];   // Sort alarm data
      statPrevSort { ExternalAccessible := 'False'; ExternalVisible := 'False'; ExternalWritable := 'False'} : Int;   // Sort on the last scan
      instProgramAlarm {InstructionName := 'Program_Alarm'; LibVersion := '1.0'; ExternalAccessible := 'False'; ExternalVisible := 'False'; ExternalWritable := 'False'} : Program_Alarm;   // Record alarm
      statAlarm { ExternalAccessible := 'False'; ExternalVisible := 'False'; ExternalWritable := 'False'} : Bool;   // Alarm is active
      statArrayFull { ExternalAccessible := 'False'; ExternalVisible := 'False'; ExternalWritable := 'False'} : Bool;   // Array is larger than MAX_AMOUNT_OF_ERRORS
      statFullRunningDowntime { ExternalAccessible := 'False'; ExternalVisible := 'False'; ExternalWritable := 'False'} : Real;   // Running downtime when array is full
      statFullPrevDowntime { ExternalAccessible := 'False'; ExternalVisible := 'False'; ExternalWritable := 'False'} : Real;   // Total downtime for all alarms not recorded in the array
   END_VAR

   VAR_TEMP 
      tempTimestamp {InstructionName := 'DTL'; LibVersion := '1.0'} : DTL;
      tempTimeErr : Int;
      tempEntryFound : Bool;
   END_VAR

   VAR CONSTANT 
      MS_TO_MIN : Real := 60000.0;   // Convert from milliseconds to minutes
   END_VAR


BEGIN
	//============================================================================================================
	// SIEMENS NV - APC Belgium
	// (c)Copyright 2018 All Rights Reserved
	//------------------------------------------------------------------------------------------------------------
	// Tested with: S7
	// -1500 with FW version V2.5, V2.6
	// Engineering: TIA Portal V15, V15.1
	// Restrictions: ---
	// Requirements: S7-1x00
	// Functionality: Pareto analysis on stop reasons
	//------------------------------------------------------------------------------------------------------------
	// Change log table:
	// Version       Date               Expert in charge        Changes applied
	// 01.00.00      14.10.2018         J.Pieters               Initial Release 
	// 02.00.00      09.05.2019         K.Bartuska              Included text, total downtime, and MTBF
	// 03.00.00      13.09.2019         K.Bartuska, M.Earnest   Included MTTR, custom sort, and continuous downtime updates         
	//============================================================================================================
	// Function : paretoAnalysis
	//============================================================================================================
	
	
	//REGION RESET_PARETO_RESULTS
	IF #statFirstScan OR (#resetPareto AND NOT #statResetParetoOld)
	THEN
	    FOR #statIndex := 1 TO "CPG_PARTEO_NO_OF_ERRORS_UPPER_LIM" DO
	        #paretoData[#statIndex].alarmID := 0;
	        #paretoData[#statIndex].percentageOccurred := 0.0;
	        #paretoData[#statIndex].timesOccurred := 0;
	        #paretoData[#statIndex].alarmMessage := '';
	        #paretoData[#statIndex].MTTR := 0.0;
	        #paretoData[#statIndex].totalDowntime := 0.0;
	    END_FOR;
	    
	    #tempTimeErr := RD_LOC_T(#statResetTimestamp);
	    #statTotalStops := 0;
	    #statTotalDowntime := 0.0;
	    #statOverallMTTR := 0.0;
	    #statFirstScan := FALSE;
	    #statPrevTotalUptime := 0.0;
	    #statStopReasonOld := 0;
	    #statArrayFull := 0;
	    #statFullPrevDowntime := 0.0;
	    
	END_IF;
	// one shot bit
	#statResetParetoOld := #resetPareto;
	//END_REGION
	
	FOR #statIndex := 1 TO "CPG_PARTEO_NO_OF_ERRORS_UPPER_LIM" DO
	    IF #paretoData[#statIndex].alarmID = #ID
	    THEN
	        #tempEntryFound := TRUE;
	    END_IF;
	END_FOR;
	
	//REGION UPDATE_DOWNTIME  
	//adjust downtime & MTTR
	
	//For a different alarm
	IF #ID <> #statStopReasonOld
	THEN
	    #statPrevTimestamp := #statCurrentTimestamp;
	    #tempTimeErr := RD_LOC_T(#statCurrentTimestamp);
	    #statBaseDowntime := 0.0;
	    #statAlarm := 0;
	    #statFullPrevDowntime := #statFullPrevDowntime + #statFullRunningDowntime;
	    #statFullRunningDowntime := 0.0;
	    
	    
	    //Update downtime when fault is active    
	ELSIF #ID = #statStopReasonOld AND #ID <> 0
	THEN
	    #tempTimeErr := RD_LOC_T(#statSameCurrentTimestamp);
	    #statAlarm := 1;
	    IF #tempEntryFound
	    THEN
	        FOR #statIndex := 1 TO "CPG_PARTEO_NO_OF_ERRORS_UPPER_LIM" DO
	            IF #paretoData[#statIndex].alarmID = #ID
	            THEN
	                #paretoData[#statIndex].totalDowntime := #statBaseDowntime + (DINT_TO_REAL(TIME_TO_DINT(T_DIFF(IN1 := #statSameCurrentTimestamp, IN2 := #statCurrentTimestamp))) / #MS_TO_MIN);
	                IF #paretoData[#statIndex].timesOccurred <> 0
	                THEN
	                    #paretoData[#statIndex].MTTR := (#paretoData[#statIndex].totalDowntime) / #paretoData[#statIndex].timesOccurred;
	                END_IF;
	                EXIT;
	            END_IF;
	        END_FOR;
	    ELSIF NOT #tempEntryFound AND #statArrayFull
	    THEN
	        #statFullRunningDowntime := DINT_TO_REAL(TIME_TO_DINT(T_DIFF(IN1 := #statSameCurrentTimestamp, IN2 := #statCurrentTimestamp))) / #MS_TO_MIN;
	    END_IF;
	END_IF;
	//END_REGION
	
	
	//REGION CREATE_PROGRAM_ALARM
	//create an alarm
	#instProgramAlarm(SIG := #statAlarm,
	               SD_1 := #ID,
	               SD_2 := #message);
	//END_REGION
	
	//REGION PARETO_MAIN
	// check if an error is active
	IF #ID <> #statStopReasonOld AND (#ID <> 0)
	THEN
	    //REGION INCREMENT_EXISTING_ALARM_ID
	    IF #tempEntryFound
	    THEN
	        FOR #statIndex := 1 TO "CPG_PARTEO_NO_OF_ERRORS_UPPER_LIM" DO
	            // find if alarm is already defined in list
	            IF #paretoData[#statIndex].alarmID = #ID
	            THEN
	                #paretoData[#statIndex].timesOccurred := #paretoData[#statIndex].timesOccurred + UINT#1;
	                EXIT; // exit this loop
	            END_IF;
	        END_FOR;
	    ELSIF NOT #tempEntryFound AND #statArrayFull
	    THEN
	        #statTotalStops := #statTotalStops + 1;
	    END_IF;
	    //END_REGION
	    
	    //REGION ADD_NEW_ALARM_ID
	    //If alarm is not defined in list then make a new entry
	    IF (NOT #tempEntryFound) AND (NOT #statArrayFull)
	    THEN
	        FOR #statIndex := 1 TO "CPG_PARTEO_NO_OF_ERRORS_UPPER_LIM" DO
	            
	            IF #paretoData[#statIndex].alarmID = 0
	            THEN
	                #paretoData[#statIndex].alarmID := #ID;
	                #paretoData[#statIndex].timesOccurred := 1;
	                #paretoData[#statIndex].alarmMessage := #message;
	                #tempEntryFound := TRUE;
	                //Array is now full
	                IF #statIndex = "CPG_PARTEO_NO_OF_ERRORS_UPPER_LIM"
	                THEN
	                    #statArrayFull := 1;
	                END_IF;
	                EXIT; // exit this loop
	            END_IF;
	        END_FOR;
	    END_IF;
	    //END_REGION
	END_IF;
	
	IF #ID <> #statStopReasonOld AND #tempEntryFound
	THEN
	    //REGION FIND_TOTAL_OCCURED_ALARMS
	    // count total number stop has occured
	    //initialize alarm counters
	    #statTotalStops := 0;
	    #statTotalDowntime := 0.0;
	    #statOverallMTTR := 0.0;
	    
	    FOR #statIndex := 1 TO "CPG_PARTEO_NO_OF_ERRORS_UPPER_LIM" DO
	        IF #paretoData[#statIndex].alarmID = #ID
	        THEN
	            #statBaseDowntime := #paretoData[#statIndex].totalDowntime;
	        END_IF;
	        IF #paretoData[#statIndex].alarmID <> 0
	        THEN
	            #statTotalStops := #statTotalStops + #paretoData[#statIndex].timesOccurred;
	            #statTotalDowntime := #statTotalDowntime + #paretoData[#statIndex].totalDowntime;
	        END_IF;
	    END_FOR;
	    
	    IF #statTotalStops <> 0
	    THEN
	        #statOverallMTTR := (#statTotalDowntime + #statFullPrevDowntime + #statFullRunningDowntime) / #statTotalStops;
	    END_IF;
	    //END_REGION
	    
	    //REGION CALCULATE_PRECENTAGE_FOR_EACH_ALARM
	    // calculate percentage each alarm occured
	    FOR #statIndex := 1 TO "CPG_PARTEO_NO_OF_ERRORS_UPPER_LIM" DO
	        IF #paretoData[#statIndex].alarmID <> 0
	        THEN
	            // avoid division by zero 
	            #paretoData[#statIndex].percentageOccurred := SEL(G := #statTotalStops <> 0,
	                                                              IN0 := 0.0,
	                                                              IN1 := ((#paretoData[#statIndex].totalDowntime) / (#statTotalDowntime + #statFullPrevDowntime + #statFullRunningDowntime)) * 100.0);
	        END_IF;
	    END_FOR;
	    //END_REGION
	END_IF;
	
	//Update downtime and MTTR when fault is still active
	IF #ID = #statStopReasonOld AND #ID <> 0
	THEN
	    //REGION FIND_TOTAL_OCCURED_ALARMS
	    IF #tempEntryFound
	    THEN
	        #statTotalDowntime := 0.0;
	        FOR #statIndex := 1 TO "CPG_PARTEO_NO_OF_ERRORS_UPPER_LIM" DO
	            #statTotalDowntime := #statTotalDowntime + #paretoData[#statIndex].totalDowntime;
	        END_FOR;
	    END_IF;
	    
	    IF #statTotalStops <> 0 THEN
	        #statOverallMTTR := (#statTotalDowntime + #statFullPrevDowntime + #statFullRunningDowntime) / #statTotalStops;
	    END_IF;
	    
	    //END_REGION
	    
	    //REGION CALCULATE_PRECENTAGE_FOR_EACH_ALARM
	    // calculate percentage each alarm occured
	    IF #tempEntryFound
	    THEN
	        FOR #statIndex := 1 TO "CPG_PARTEO_NO_OF_ERRORS_UPPER_LIM" DO
	            IF #paretoData[#statIndex].alarmID <> 0
	            THEN
	                // avoid division by zero 
	                #paretoData[#statIndex].percentageOccurred := SEL(G := #statTotalStops <> 0,
	                                                                  IN0 := 0.0,
	                                                                  IN1 := ((#paretoData[#statIndex].totalDowntime) / (#statTotalDowntime + #statFullPrevDowntime + #statFullRunningDowntime)) * 100.0);
	            END_IF;
	        END_FOR;
	    END_IF;
	    //END_REGION
	END_IF;
	
	//Sort the alarm array
	//REGION SORT_ARRAY_CRITERIA
	IF #sort = 0 THEN
	    #statSort := 'totalDowntime';
	ELSIF #sort = 1 THEN
	    #statSort := 'percentageOccurred';
	ELSIF #sort = 2 THEN
	    #statSort := 'timesOccurred';
	ELSIF #sort = 3 THEN
	    #statSort := 'MTTR';
	END_IF;
	
	// Sort list: most [statSort] alarms on top (index 1)
	IF #statPrevSort <> #sort OR #ID <> #statStopReasonOld
	THEN
	    #instShellSortPareto(mode := TRUE,
	                        sortBy := #statSort,
	                        variantArray := #paretoData);
	END_IF;
	#statPrevSort := #sort;
	//END_REGION
	
	#statStopReasonOld := #ID;
	//END_REGION
	
	//REGION SET_OUTPUTS
	//set other outputs
	#totalStops := #statTotalStops;
	#totalDowntime := #statTotalDowntime + #statFullPrevDowntime + #statFullRunningDowntime;
	#MTTR := #statOverallMTTR;
	
	//compute total shift time, the amount and percent the machine was up
	#tempTimeErr := RD_LOC_T(#tempTimestamp);
	#totalTimeSinceReset := DINT_TO_REAL(TIME_TO_DINT(T_DIFF(IN1 := #tempTimestamp, IN2 := #statResetTimestamp))) / #MS_TO_MIN;
	
	#totalUptime := 0.0;
	
	//if a fault is active the uptime should stay at its previous value
	IF #ID = 0 THEN
	    #totalUptime := #totalTimeSinceReset - (#statTotalDowntime + #statFullPrevDowntime + #statFullRunningDowntime);
	    #statPrevTotalUptime := #totalUptime;
	ELSE
	    #totalUptime := #statPrevTotalUptime;
	END_IF;
	
	//avoid dividing by zero
	IF #statTotalStops = 0 THEN
	    #MTBF := #totalUptime;
	ELSE
	    #MTBF := #totalUptime / #statTotalStops;
	END_IF;
	
	#percentUptime := 100.0 * (#totalUptime) / (#totalTimeSinceReset);
	//END_REGION
	
	
	//  -------------- END OF LOGIC -------------------------
	ENO := TRUE;   // Set the ENO output
END_FUNCTION_BLOCK

FUNCTION_BLOCK "CPG_ShellSortPareto"
TITLE = CPG_ShellSortPareto
{ S7_Optimized_Access := 'TRUE' }
AUTHOR : 'tech.team.motioncontrol@siemens.com'
FAMILY : CPG
VERSION : 1.1
//Support: tech.team.motioncontrol@siemens.com
   VAR_INPUT 
      mode { ExternalAccessible := 'False'; ExternalVisible := 'False'; ExternalWritable := 'False'} : Bool;   // True = sort decending, false = sort ascending
      sortBy { ExternalAccessible := 'False'; ExternalVisible := 'False'; ExternalWritable := 'False'} : String[30];   // Sorting method
   END_VAR

   VAR_OUTPUT 
      done { ExternalAccessible := 'False'; ExternalVisible := 'False'; ExternalWritable := 'False'} : Bool;   // Sort completed
      error { ExternalAccessible := 'False'; ExternalVisible := 'False'; ExternalWritable := 'False'} : Bool;   // Error while sorting
      statusID { ExternalAccessible := 'False'; ExternalVisible := 'False'; ExternalWritable := 'False'} : UInt;   // Indicates block in which error occurred
      status { ExternalAccessible := 'False'; ExternalVisible := 'False'; ExternalWritable := 'False'} : Word;   // Status word
   END_VAR

   VAR_IN_OUT 
      variantArray : Variant;   // Array to be sorted
   END_VAR

   VAR 
      statOptions { ExternalAccessible := 'False'; ExternalVisible := 'False'; ExternalWritable := 'False'} : Struct   // Options for sorting alarm array
         totalDowntime { ExternalAccessible := 'False'; ExternalVisible := 'False'; ExternalWritable := 'False'} : String[30] := 'totalDowntime';
         timesOccurred { ExternalAccessible := 'False'; ExternalVisible := 'False'; ExternalWritable := 'False'} : String[30] := 'timesOccurred';
         MTTR { ExternalAccessible := 'False'; ExternalVisible := 'False'; ExternalWritable := 'False'} : String[30] := 'MTTR';
         percentageOccurred { ExternalAccessible := 'False'; ExternalVisible := 'False'; ExternalWritable := 'False'} : String[30] := 'percentageOccurred';
      END_STRUCT;
   END_VAR

   VAR_TEMP 
      tempArrayPareto : Array[1.."CPG_PARTEO_NO_OF_ERRORS_UPPER_LIM"] of "CPG_typePareto";
      tempElementCount : Int;
      tempElementCopyCount : UDInt;
      tempMoveBlkError : Int;
      tempIncrement : Int;
      tempForCounter : Int;
      tempExchangeIndex : Int;
      tempExchangeVariable : "CPG_typePareto";
      tempTypeTag : "CPG_typePareto";
   END_VAR

   VAR CONSTANT 
      MAX_ARRAY_ELEMENTS : Int := 1000;
      NO_ERROR : Word := 16#0000;
      NO_CURRENT_JOBS : Word := 16#7000;
      EMPTY_ARRAY : Word := 16#8200;
      NOT_AN_ARRAY : Word := 16#8201;
      WRONG_ELEMENT_TYPE : Word := 16#8202;
      TOO_MANY_ELEMENTS : Word := 16#8203;
      ERROR_IN_THIS_BLOCK : UInt := 1;
      ERROR_MOVE_BLK_VARIANT_R : UInt := 2;
      ERROR_MOVE_BLK_VARIANT_W : UInt := 3;
   END_VAR


BEGIN
	//=============================================================================
	// SIEMENS AG
	// (c)Copyright 2017
	//-----------------------------------------------------------------------------
	// Library:       LGF (Library General Functions)
	// Tested with:   CPU1212C DC/DC/DC FW:V4.2
	// Engineering:   TIA Portal V14 Update 1
	// Restrictions:  -
	// Requirements:  PLC (S7-1200 / S7-1500)
	// Functionality: A shellsort algorithm with a complexity between 'n^2' and
	//                'n log n' for average, best and worst case inputs and space
	//                complexity '1'.
	//                The block accepts a pareto array as an inOut-variable and
	//                returns the sorted version of the array in the same variable
	//-----------------------------------------------------------------------------
	// Change log table:
	// Version  Date        Expert in charge / Changes applied
	// 01.00.00 19.08.2015  Siemens Industry Online Support
	//                      First released version
	// 01.01.00 19.05.2016  Siemens Industry Online Support
	//                      New function: reverse sort
	// 01.01.01 02.01.2017  Siemens Industry Online Support
	//                      Upgrade: TIA Portal V14 Update 1
	// 01.01.02 17.08.2018  Siemens Industry Online Support
	//                      Upgrade: TIA V15 Update 2
	// 01.01.03 26.10.2018  APC-BE - Pieters
	//                      Modified for use with pareto type
	// 01.01.03 13.09.2019  Modified with variable sort parameters                  
	//-----------------------------------------------------------------------------
	//Status Codes:
	// 16#7000:  No current jobs
	// 16#0000:  Job finished; Note: There is no "Busy"-Status because the block is
	//           finished within a single cycle
	// 16#8200:  Error: Parameter is an array with only one element
	// 16#8201:  Error: Parameter is not an array
	// 16#8202:  Error: Parameter is an array of the wrong type
	//           (correct type is Real)
	// 16#8203:  Error: There are too many Elements in the array
	//           (default: max. 1000 Elements)
	//=============================================================================
	
	// Change note: If you wish to use this shellsort block for other datatypes,
	// you simply need to change the following variables to that type
	// 1. tempExchangeVariable
	// 2. tempTypeTag
	// 3. tempArray<Type>
	// Space note: If you wish to reduce the space of this block, you may reduce the
	// size of the tempArray<Type> to one just big enough for your specific purpose
	// It is not recommended to increase the size significantly.
	
	// Initialization
	#tempElementCount := 0;
	#tempElementCopyCount := 0;
	#tempMoveBlkError := 0;
	#tempIncrement := 0;
	#tempForCounter := 0;
	#tempExchangeIndex := 0;
	#tempExchangeVariable.alarmID := 0;
	#tempExchangeVariable.percentageOccurred := 0.0;
	#tempExchangeVariable.timesOccurred := 0;
	#tempTypeTag.alarmID := 0;
	#tempTypeTag.percentageOccurred := 0.0;
	#tempTypeTag.timesOccurred := 0;
	
	// Set "No current job" status
	#done := false;
	#error := false;
	#statusID := #ERROR_IN_THIS_BLOCK;
	#status := #NO_CURRENT_JOBS;
	
	
	// If the variant inOut-parameter is not an array, set error status 8201
	IF (IS_ARRAY(#variantArray) = false) THEN
	    #error := true;
	    #statusID := #ERROR_IN_THIS_BLOCK;
	    #status := #NOT_AN_ARRAY;
	    RETURN;
	ELSE
	    IF TypeOfElements(#variantArray) = TypeOf(#tempTypeTag) THEN
	        // If the parameter is an array of the type real, get the element count
	        #tempElementCopyCount := CountOfElements(#variantArray);
	        #tempElementCount := UDINT_TO_INT(CountOfElements(#variantArray));
	        // Check whether the variant array contains less than the maximum possible amount of elements
	        IF #tempElementCount > #MAX_ARRAY_ELEMENTS THEN
	            #error := true;
	            #statusID := #ERROR_IN_THIS_BLOCK;
	            #status := #TOO_MANY_ELEMENTS;
	            RETURN;
	        END_IF;
	    ELSE
	        // If the parameter is an array but not of the type real, set an error status
	        #error := true;
	        #statusID := #ERROR_IN_THIS_BLOCK;
	        #status := #WRONG_ELEMENT_TYPE;
	        RETURN;
	    END_IF;
	END_IF;
	
	// If there are more than zero elements to sort, begin sorting    
	IF #tempElementCount > 1 AND #error = false THEN
	    
	    // Read the elements of the incoming variant-array and write into the local array
	    #tempMoveBlkError := MOVE_BLK_VARIANT(COUNT := #tempElementCopyCount,
	                                          DEST => #tempArrayPareto,
	                                          DEST_INDEX := 0,
	                                          SRC := #variantArray,
	                                          SRC_INDEX := 0);
	    
	    // Error handling for MOVE_BLK_VARIANT
	    IF #tempMoveBlkError <> 0 THEN
	        #error := true;
	        #statusID := #ERROR_MOVE_BLK_VARIANT_R;
	        #status := INT_TO_WORD(#tempMoveBlkError);
	        RETURN;
	    END_IF;
	    
	    // ShellSort Start
	    #tempIncrement := 1;
	    REPEAT
	        #tempIncrement := (3 * #tempIncrement) + 1;
	    UNTIL #tempIncrement > #tempElementCount
	    END_REPEAT;
	    
	    REPEAT
	        #tempIncrement := DINT_TO_INT(TRUNC(#tempIncrement / 3));
	        FOR #tempForCounter := (#tempIncrement + 1) TO #tempElementCount DO
	            #tempExchangeVariable := #tempArrayPareto[#tempForCounter];
	            #tempExchangeIndex := #tempForCounter;
	            
	            IF #mode  // Modification Version 02.00.00
	            THEN      //mode = TRUE --> sort descending  
	                //Downtime
	                IF #sortBy = #statOptions.totalDowntime THEN
	                    WHILE ((#tempArrayPareto[#tempExchangeIndex - #tempIncrement].totalDowntime < #tempExchangeVariable.totalDowntime)) DO
	                        #tempArrayPareto[#tempExchangeIndex] := #tempArrayPareto[#tempExchangeIndex - #tempIncrement];
	                        #tempExchangeIndex := #tempExchangeIndex - #tempIncrement;
	                        IF (#tempExchangeIndex <= #tempIncrement) THEN
	                            GOTO EXITWhile;
	                        END_IF;
	                    END_WHILE;
	                    //Times Occurred    
	                ELSIF #sortBy = #statOptions.timesOccurred THEN
	                    WHILE ((#tempArrayPareto[#tempExchangeIndex - #tempIncrement].timesOccurred < #tempExchangeVariable.timesOccurred)) DO
	                        #tempArrayPareto[#tempExchangeIndex] := #tempArrayPareto[#tempExchangeIndex - #tempIncrement];
	                        #tempExchangeIndex := #tempExchangeIndex - #tempIncrement;
	                        IF (#tempExchangeIndex <= #tempIncrement) THEN
	                            GOTO EXITWhile;
	                        END_IF;
	                    END_WHILE;
	                    //Percentage Occurred
	                ELSIF #sortBy = #statOptions.percentageOccurred THEN
	                    WHILE ((#tempArrayPareto[#tempExchangeIndex - #tempIncrement].percentageOccurred < #tempExchangeVariable.percentageOccurred)) DO
	                        #tempArrayPareto[#tempExchangeIndex] := #tempArrayPareto[#tempExchangeIndex - #tempIncrement];
	                        #tempExchangeIndex := #tempExchangeIndex - #tempIncrement;
	                        IF (#tempExchangeIndex <= #tempIncrement) THEN
	                            GOTO EXITWhile;
	                        END_IF;
	                    END_WHILE;
	                    // MTTR
	                ELSIF #sortBy = #statOptions.MTTR THEN
	                    WHILE ((#tempArrayPareto[#tempExchangeIndex - #tempIncrement].MTTR < #tempExchangeVariable.MTTR)) DO
	                        #tempArrayPareto[#tempExchangeIndex] := #tempArrayPareto[#tempExchangeIndex - #tempIncrement];
	                        #tempExchangeIndex := #tempExchangeIndex - #tempIncrement;
	                        IF (#tempExchangeIndex <= #tempIncrement) THEN
	                            GOTO EXITWhile;
	                        END_IF;
	                    END_WHILE;
	                END_IF;
	                
	            ELSE      // mode = FALSE --> sort ascending
	                WHILE ((#tempArrayPareto[#tempExchangeIndex - #tempIncrement].MTTR > #tempExchangeVariable.MTTR)) DO
	                    #tempArrayPareto[#tempExchangeIndex] := #tempArrayPareto[#tempExchangeIndex - #tempIncrement];
	                    #tempExchangeIndex := #tempExchangeIndex - #tempIncrement;
	                    IF (#tempExchangeIndex <= #tempIncrement) THEN
	                        GOTO EXITWhile;
	                    END_IF;
	                END_WHILE;
	            END_IF;
	            
	        EXITWhile:
	            #tempArrayPareto[#tempExchangeIndex] := #tempExchangeVariable;
	        END_FOR;
	    UNTIL #tempIncrement <= 1
	    END_REPEAT;
	    // ShellSort End
	    
	    // Write the elements of the local array back to the variant array
	    #tempMoveBlkError := MOVE_BLK_VARIANT(COUNT := #tempElementCopyCount,
	                                          DEST => #variantArray,
	                                          DEST_INDEX := 0,
	                                          SRC := #tempArrayPareto,
	                                          SRC_INDEX := 0);
	    
	    // Error handling for MOVE_BLK_VARIANT
	    IF #tempMoveBlkError <> 0 THEN
	        #statusID := #ERROR_MOVE_BLK_VARIANT_W;
	        #status := INT_TO_WORD(#tempMoveBlkError);
	        RETURN;
	    END_IF;
	    
	    // Set output status = "Job Finished" and output Done = true
	    #done := true;
	    #status := #NO_ERROR;
	    
	ELSIF #tempElementCount <= 1 THEN
	    // If there are 0 elements in the array, set status to "Error: Parameter is an empty array"
	    #error := true;
	    #statusID := #ERROR_IN_THIS_BLOCK;
	    #status := #EMPTY_ARRAY;
	END_IF;
	
	//  -------------- END OF LOGIC -------------------------
	ENO := TRUE;   // Set the ENO output
END_FUNCTION_BLOCK

FUNCTION_BLOCK "UN_06_MiscFunctions"   // FB31626, LAD
TITLE = UN_06_MiscFunctions
{ S7_Optimized_Access := 'TRUE' }
AUTHOR : tech.team.motioncontrol@siemens.com
FAMILY : CPG
VERSION : 1.1
// Support: tech.team.motioncontrol@siemens.com
// stored: AutoNumber true, IsIECCheckEnabled false, IsRetainMemResEnabled false, MemoryReserve 100, SetENOAutomatically false, UDAEnableTagReadback false
   VAR
      instOEE_Calculation { ExternalAccessible := 'False'; ExternalVisible := 'False'; ExternalWritable := 'False'; S7_SetPoint := 'True'} : "CPG_OEE";   // FB used to calculate the real-time OEE value
      statOneShot_ProdConsumerCounter { ExternalAccessible := 'False'; ExternalVisible := 'False'; ExternalWritable := 'False'} : Bool;   // One Shot - products consumed counter
      statOneShot_ProdProcessedCounter { ExternalAccessible := 'False'; ExternalVisible := 'False'; ExternalWritable := 'False'} : Bool;   // One Shot - products processed counter
      statOneShot_ProdDefectiveCounter { ExternalAccessible := 'False'; ExternalVisible := 'False'; ExternalWritable := 'False'} : Bool;   // One Shot - products defective counter
   END_VAR
   VAR_TEMP
      tempReadClockRetVal : Int;
      tempProductionCounterTrigger : Bool;
   END_VAR
   VAR_TEMP   // added for the SCL form of the ladder/FBD networks
      _w1 : Bool;
   END_VAR
BEGIN

REGION Network 1: Update the PackTags Admin.PLC_Date_Time with current PLC time
   // 1) Update the "PackTags".Admin.PLC_Date_Time with the current PLC time.
   // 2) Update "HMI_Data".PLC_Date_Time.DATE_TIME with current PLC time so the HMI 
   // and PLC are time synchronized.
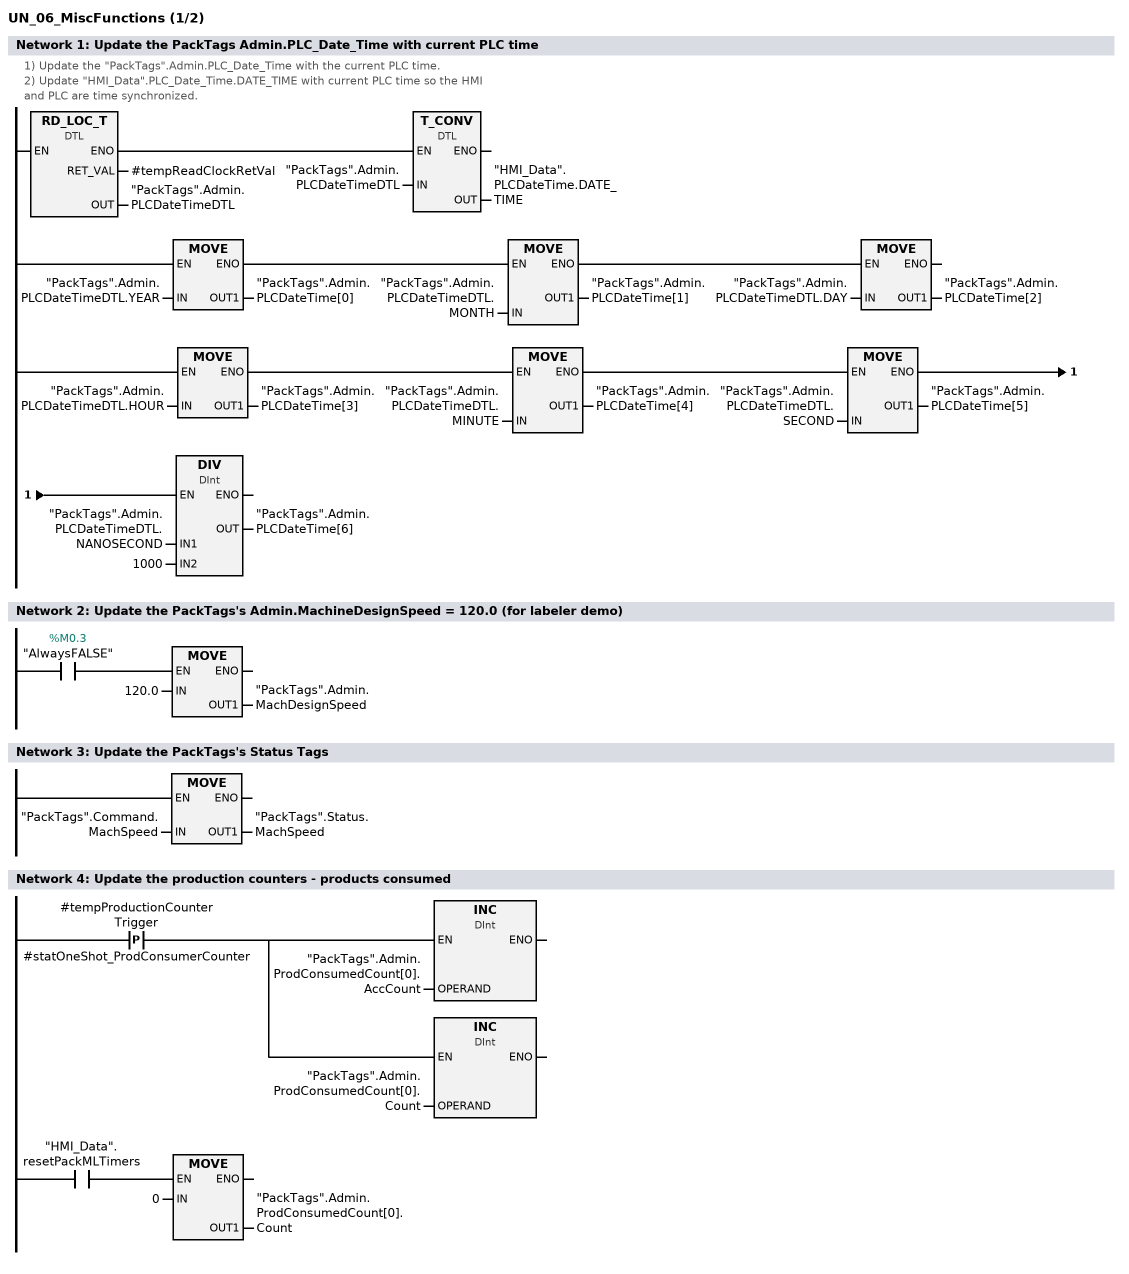
   RUNG wire#powerrail
      { S7_Templates := "date_type := DTL" } RD_LOC_T(RET_VAL => #tempReadClockRetVal, OUT => "PackTags".Admin.PLCDateTimeDTL)
      { S7_Templates := "[src_type := DTL, dest_type := Date_And_Time]" } T_CONV(IN := "PackTags".Admin.PLCDateTimeDTL, OUT => "HMI_Data".PLCDateTime.DATE_TIME)
   END_RUNG
   RUNG wire#powerrail
      Move(in := "PackTags".Admin.PLCDateTimeDTL.YEAR, out1 => "PackTags".Admin.PLCDateTime[0])
      Move(in := "PackTags".Admin.PLCDateTimeDTL.MONTH, out1 => "PackTags".Admin.PLCDateTime[1])
      Move(in := "PackTags".Admin.PLCDateTimeDTL.DAY, out1 => "PackTags".Admin.PLCDateTime[2])
   END_RUNG
   RUNG wire#powerrail
      Move(in := "PackTags".Admin.PLCDateTimeDTL.HOUR, out1 => "PackTags".Admin.PLCDateTime[3])
      Move(in := "PackTags".Admin.PLCDateTimeDTL.MINUTE, out1 => "PackTags".Admin.PLCDateTime[4])
      Move(in := "PackTags".Admin.PLCDateTimeDTL.SECOND, out1 => "PackTags".Admin.PLCDateTime[5])
      { S7_Templates := "SrcType := DInt" } Div(in1 := "PackTags".Admin.PLCDateTimeDTL.NANOSECOND, in2 := 1000, out => "PackTags".Admin.PLCDateTime[6])
   END_RUNG
   // the same network as SCL:
   #tempReadClockRetVal := RD_LOC_T(OUT => "PackTags".Admin.PLCDateTimeDTL, ENO => #_w1);
   IF #_w1 THEN
       T_CONV(IN := "PackTags".Admin.PLCDateTimeDTL, OUT => "HMI_Data".PLCDateTime.DATE_TIME);
   END_IF;
   "PackTags".Admin.PLCDateTime[0] := "PackTags".Admin.PLCDateTimeDTL.YEAR;
   "PackTags".Admin.PLCDateTime[1] := "PackTags".Admin.PLCDateTimeDTL.MONTH;
   "PackTags".Admin.PLCDateTime[2] := "PackTags".Admin.PLCDateTimeDTL.DAY;
   "PackTags".Admin.PLCDateTime[3] := "PackTags".Admin.PLCDateTimeDTL.HOUR;
   "PackTags".Admin.PLCDateTime[4] := "PackTags".Admin.PLCDateTimeDTL.MINUTE;
   "PackTags".Admin.PLCDateTime[5] := "PackTags".Admin.PLCDateTimeDTL.SECOND;
   "PackTags".Admin.PLCDateTime[6] := "PackTags".Admin.PLCDateTimeDTL.NANOSECOND / 1000;
END_REGION

REGION Network 2: Update the PackTags's Admin.MachineDesignSpeed = 120.0 (for labeler demo)
   RUNG wire#powerrail
      Contact( "AlwaysFALSE" )
      Move(in := 120.0, out1 => "PackTags".Admin.MachDesignSpeed)
   END_RUNG
   // the same network as SCL:
   IF "AlwaysFALSE" THEN "PackTags".Admin.MachDesignSpeed := 120.0; END_IF;
END_REGION

REGION Network 3: Update the PackTags's Status Tags
   RUNG wire#powerrail
      Move(in := "PackTags".Command.MachSpeed, out1 => "PackTags".Status.MachSpeed)
   END_RUNG
   // the same network as SCL:
   "PackTags".Status.MachSpeed := "PackTags".Command.MachSpeed;
END_REGION

REGION Network 4: Update the production counters - products consumed
   RUNG wire#powerrail
      P_Contact(operand := #tempProductionCounterTrigger, bit := #statOneShot_ProdConsumerCounter)
      wire#w1
      { S7_Templates := "DestType := DInt" } Inc( "PackTags".Admin.ProdConsumedCount[0].AccCount )
   END_RUNG
   RUNG wire#w1
      { S7_Templates := "DestType := DInt" } Inc( "PackTags".Admin.ProdConsumedCount[0].Count )
   END_RUNG
   RUNG wire#powerrail
      Contact( "HMI_Data".resetPackMLTimers )
      Move(in := 0, out1 => "PackTags".Admin.ProdConsumedCount[0].Count)
   END_RUNG
   // the same network as SCL:
   #_w1 := #tempProductionCounterTrigger AND NOT #statOneShot_ProdConsumerCounter;   // rising edge of #tempProductionCounterTrigger
   #statOneShot_ProdConsumerCounter := #tempProductionCounterTrigger;
   IF #_w1 THEN
       "PackTags".Admin.ProdConsumedCount[0].AccCount := "PackTags".Admin.ProdConsumedCount[0].AccCount + 1;
       "PackTags".Admin.ProdConsumedCount[0].Count := "PackTags".Admin.ProdConsumedCount[0].Count + 1;
   END_IF;
   IF "HMI_Data".resetPackMLTimers THEN "PackTags".Admin.ProdConsumedCount[0].Count := 0; END_IF;
END_REGION

REGION Network 5: Update the production counters - products processed
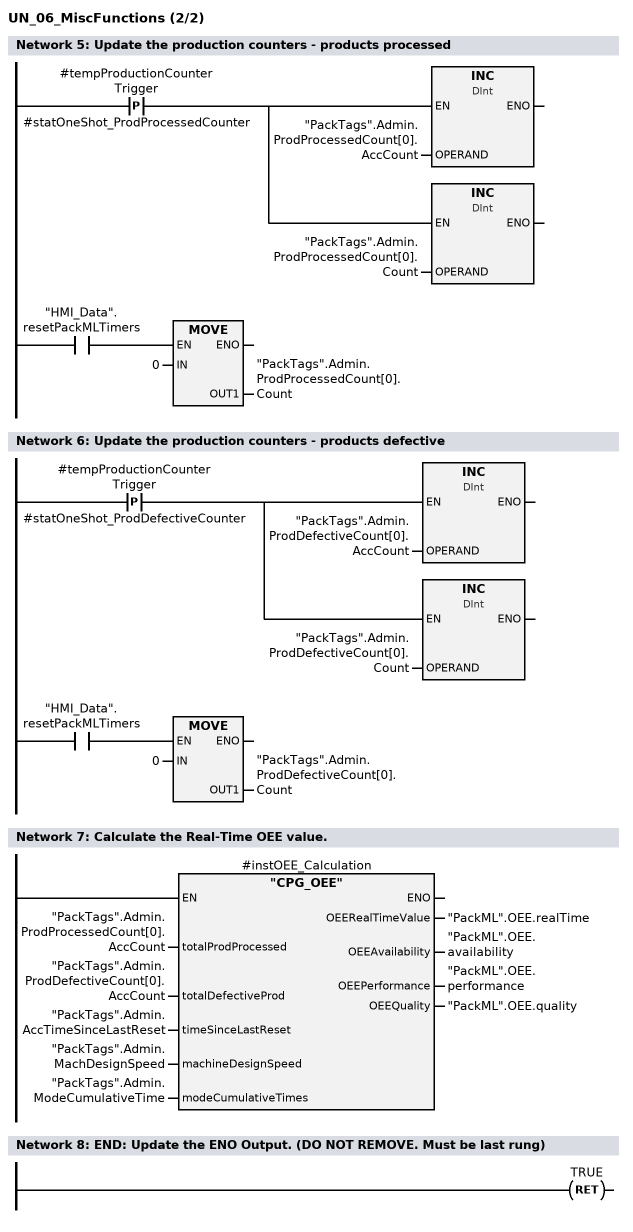
   RUNG wire#powerrail
      P_Contact(operand := #tempProductionCounterTrigger, bit := #statOneShot_ProdProcessedCounter)
      wire#w1
      { S7_Templates := "DestType := DInt" } Inc( "PackTags".Admin.ProdProcessedCount[0].AccCount )
   END_RUNG
   RUNG wire#w1
      { S7_Templates := "DestType := DInt" } Inc( "PackTags".Admin.ProdProcessedCount[0].Count )
   END_RUNG
   RUNG wire#powerrail
      Contact( "HMI_Data".resetPackMLTimers )
      Move(in := 0, out1 => "PackTags".Admin.ProdProcessedCount[0].Count)
   END_RUNG
   // the same network as SCL:
   #_w1 := #tempProductionCounterTrigger AND NOT #statOneShot_ProdProcessedCounter;   // rising edge of #tempProductionCounterTrigger
   #statOneShot_ProdProcessedCounter := #tempProductionCounterTrigger;
   IF #_w1 THEN
       "PackTags".Admin.ProdProcessedCount[0].AccCount := "PackTags".Admin.ProdProcessedCount[0].AccCount + 1;
       "PackTags".Admin.ProdProcessedCount[0].Count := "PackTags".Admin.ProdProcessedCount[0].Count + 1;
   END_IF;
   IF "HMI_Data".resetPackMLTimers THEN "PackTags".Admin.ProdProcessedCount[0].Count := 0; END_IF;
END_REGION

REGION Network 6: Update the production counters - products defective
   RUNG wire#powerrail
      P_Contact(operand := #tempProductionCounterTrigger, bit := #statOneShot_ProdDefectiveCounter)
      wire#w1
      { S7_Templates := "DestType := DInt" } Inc( "PackTags".Admin.ProdDefectiveCount[0].AccCount )
   END_RUNG
   RUNG wire#w1
      { S7_Templates := "DestType := DInt" } Inc( "PackTags".Admin.ProdDefectiveCount[0].Count )
   END_RUNG
   RUNG wire#powerrail
      Contact( "HMI_Data".resetPackMLTimers )
      Move(in := 0, out1 => "PackTags".Admin.ProdDefectiveCount[0].Count)
   END_RUNG
   // the same network as SCL:
   #_w1 := #tempProductionCounterTrigger AND NOT #statOneShot_ProdDefectiveCounter;   // rising edge of #tempProductionCounterTrigger
   #statOneShot_ProdDefectiveCounter := #tempProductionCounterTrigger;
   IF #_w1 THEN
       "PackTags".Admin.ProdDefectiveCount[0].AccCount := "PackTags".Admin.ProdDefectiveCount[0].AccCount + 1;
       "PackTags".Admin.ProdDefectiveCount[0].Count := "PackTags".Admin.ProdDefectiveCount[0].Count + 1;
   END_IF;
   IF "HMI_Data".resetPackMLTimers THEN "PackTags".Admin.ProdDefectiveCount[0].Count := 0; END_IF;
END_REGION

REGION Network 7: Calculate the Real-Time OEE value.
   RUNG wire#powerrail
      #instOEE_Calculation(totalProdProcessed := "PackTags".Admin.ProdProcessedCount[0].AccCount, totalDefectiveProd := "PackTags".Admin.ProdDefectiveCount[0].AccCount, timeSinceLastReset := "PackTags".Admin.AccTimeSinceLastReset, machineDesignSpeed := "PackTags".Admin.MachDesignSpeed, modeCumulativeTimes := "PackTags".Admin.ModeCumulativeTime, OEERealTimeValue => "PackML".OEE.realTime, OEEAvailability => "PackML".OEE.availability, OEEPerformance => "PackML".OEE.performance, OEEQuality => "PackML".OEE.quality)
   END_RUNG
   // the same network as SCL:
   #instOEE_Calculation(totalProdProcessed := "PackTags".Admin.ProdProcessedCount[0].AccCount,   // "CPG_OEE"
                        totalDefectiveProd := "PackTags".Admin.ProdDefectiveCount[0].AccCount,
                        timeSinceLastReset := "PackTags".Admin.AccTimeSinceLastReset,
                        machineDesignSpeed := "PackTags".Admin.MachDesignSpeed,
                        modeCumulativeTimes := "PackTags".Admin.ModeCumulativeTime,
                        OEERealTimeValue => "PackML".OEE.realTime,
                        OEEAvailability => "PackML".OEE.availability,
                        OEEPerformance => "PackML".OEE.performance,
                        OEEQuality => "PackML".OEE.quality);
END_REGION

REGION Network 8: END: Update the ENO Output. (DO NOT REMOVE. Must be last rung)
   RUNG wire#powerrail
      ReturnCoil( TRUE )
   END_RUNG
   // the same network as SCL:
   ENO := TRUE;
   RETURN;
END_REGION
END_FUNCTION_BLOCK

FUNCTION_BLOCK "CPG_OEE"
TITLE = CPG_OEE
{ S7_Optimized_Access := 'TRUE' }
AUTHOR : 'tech.team.motioncontrol@siemens.com'
FAMILY : CPG
VERSION : 1.0
//Support: tech.team.motioncontrol@siemens.com
   VAR_INPUT 
      totalProdProcessed { ExternalAccessible := 'False'; ExternalVisible := 'False'; ExternalWritable := 'False'} : DInt;   // Total Number OF Products Processed
      totalDefectiveProd { ExternalAccessible := 'False'; ExternalVisible := 'False'; ExternalWritable := 'False'} : DInt;   // Total Number OF Defective Products
      timeSinceLastReset { ExternalAccessible := 'False'; ExternalVisible := 'False'; ExternalWritable := 'False'} : DInt;   // Total Acumulative TIME since Last RESET
      machineDesignSpeed { ExternalAccessible := 'False'; ExternalVisible := 'False'; ExternalWritable := 'False'} : Real;   // Machine Design Speed
   END_VAR

   VAR_OUTPUT 
      OEERealTimeValue { ExternalAccessible := 'False'; ExternalVisible := 'False'; ExternalWritable := 'False'} : Real;   // REAL TIME OEE value (availabilty x performance x quality)
      OEEAvailability { ExternalAccessible := 'False'; ExternalVisible := 'False'; ExternalWritable := 'False'} : Real;   // OEE - Availability value
      OEEPerformance { ExternalAccessible := 'False'; ExternalVisible := 'False'; ExternalWritable := 'False'} : Real;   // OEE - Performance value
      OEEQuality { ExternalAccessible := 'False'; ExternalVisible := 'False'; ExternalWritable := 'False'} : Real;   // OEE - Quality  value
   END_VAR

   VAR_IN_OUT 
      modeCumulativeTimes : Array[0.."LPMLV30_MODES_UPPER_LIM"] of DInt;   // Mode Cummulative Times
   END_VAR

   VAR 
      statTotalProdProcessed_In { ExternalAccessible := 'False'; ExternalVisible := 'False'; ExternalWritable := 'False'} : DInt;   // Initial "TotalProdProcessed" value after accum TIME reset
      statTotalDefectiveProd_In { ExternalAccessible := 'False'; ExternalVisible := 'False'; ExternalWritable := 'False'} : DInt;   // Initial "TotalDefectiveProcessed" value after accum TIME reset
      statAcumTimeEqualZero { ExternalAccessible := 'False'; ExternalVisible := 'False'; ExternalWritable := 'False'} : Bool;   // The "TimeSinceLastReset" is = 0 seconds
      statAcumTimeEqualZeroOS { ExternalAccessible := 'False'; ExternalVisible := 'False'; ExternalWritable := 'False'} : Bool;   // OneShot for "TimeSinceLastReset" is = 0 seconds
   END_VAR

   VAR_TEMP 
      tempTimeSinceLastReset : Real;   // used to eliminate divide by zero errors
      tempTotalProducts : Real;   // used to eliminate divide by zero errors
      tempDefectiveProducts : Real;   // used to eliminate divide by zero errors
   END_VAR


BEGIN
	//============================================================================================================
	// SIEMENS AG
	// (c)Copyright 2018 All Rights Reserved
	//------------------------------------------------------------------------------------------------------------
	// Project: CPG Template
	// Tested with: S7-1500 with FW version V2.1
	// Engineering: TIA Portal V14
	// Restrictions: ---
	// Requirements: S7-1500
	// Functionality:  calculate real-time OEE values
	// Support: tech.team.motioncontrol@siemens.com
	//------------------------------------------------------------------------------------------------------------
	// Change log table:
	// Version       Date               Expert in charge    Changes applied
	//  01.00.00     28.02.1012         MP                  Original - using OEE Realtime calculation
	//  01.01.00     04.09.2014         MP                  Added seperate Availabity, Performace, Quality calculation
	//  01.02.00     07.07.2014         MP                  Updated interface FOR new Mode/State FB          
	//  01.02.01     01.02.2016         MP                  Added logic to prevent floating point / divide by zero errors
	//  02.00.00     01.01.2018         MP                  Prepared for CPG Release
	//  02.01.00     29.05.2018         JP                  Adopted to styleguide
	//============================================================================================================
	// Function Block : CPG_OEE
	//============================================================================================================
	
	// ===========================================================================
	//  Begin the LOGIC section:
	//  
	(* ISA TR88.00.02 Document - 9.1 OEE Definition:
	Overall Equipment Effectiveness (OEE) is a measure comparing how well manufacturing equipment is running compared to the ideal plant. The resulting measurement is expressed as the ratio of the actual
	output of the equipment divided by the maximum possible output of the equipment under ideal conditions. OEE is calculated by multiplying three independently measured values: Availability,
	Performance Rate, and Quality Rate. The fundamental OEE definition is defined as an availability ratio multiplied by a performance ratio multiplied by a quality ratio.
	
	OEE = Availability x Performance x Quality
	
	Where each component is defined as the following:
	Availability = Operating Time / Planned Production Time
	Performance = Total Pieces / (Operating Time* Ideal Run Rate)
	Quality = Good Pieces / Total Pieces
	
	OEE is often displayed as a waterfall object in which the major components of Availability, Performance, and Quality are displayed graphically.
	*)
	
	// Determine is TimeSinceLastReset value is equal to zero.
	IF  #timeSinceLastReset   = 0 THEN
	    #statAcumTimeEqualZero   := TRUE;  // SET the AcumTimeEqualZero bool tag
	ELSE
	    #statAcumTimeEqualZero   := FALSE; // RESET the AcumTimeEqualZero bool tag
	    #statAcumTimeEqualZeroOS := FALSE; // RESET the AcumTimeEqualZero one-shot bool tag
	END_IF;
	
	// Update the AcumTimeEqualZeroOS One-Shot bool
	IF #statAcumTimeEqualZero AND NOT #statAcumTimeEqualZeroOS THEN
	   #statAcumTimeEqualZeroOS := TRUE;  // Set the One-Shot bool tag
	END_IF;
	
	// Update the initial product count values after the accum timer value has been reset
	IF #statAcumTimeEqualZeroOS THEN
	   #statTotalProdProcessed_In := #totalProdProcessed;
	   #statTotalDefectiveProd_In := #totalDefectiveProd;
	END_IF;  
	
	// Update the TimeSinceLastReset temp. value.  If = 0 (zero) then change to 0.0001 to ensure no divide by zero errors
	IF #timeSinceLastReset = 0 THEN
	    #tempTimeSinceLastReset := 0.0001;
	ELSE
	    #tempTimeSinceLastReset := DINT_TO_REAL(#timeSinceLastReset);
	END_IF;
	
	
	
	(*  9.1.1 Availability Definition
	Availability is defined as operating time divided by planned production time. The basic concept behind availability is to show the time the machine has been running divided by the time that the
	machine has been planned to run. Typical losses in this area are losses to unplanned maintenance, cleaning, changeovers, and breakdowns.
	* Availability = Operating Time / Planned Production Time Operating Time is defined as the amount of time the machine has been attempting to produce parts.  
	* Planned Production Time is defined as the total amount of time the machine has been scheduled to run. 
	*)
	// Availablity = operating time (attempt to run production) / planned production time
	#OEEAvailability :=   DINT_TO_REAL (#modeCumulativeTimes[1]) / #tempTimeSinceLastReset;
	IF #OEEAvailability > 1.0 THEN #OEEAvailability := 1.0; END_IF;
	IF #OEEAvailability < 0.0 THEN #OEEAvailability := 0.0; END_IF;
	
	(* 9.1.2 Performance Definition
	Performance is defined as the total number of pieces on which the machine operated divided by the ideal production if a machine ran perfectly for the allocated amount of operating time.
	* Performance = Total Pieces / (Operating Time* Ideal Run Rate).  
	* Total Pieces is defined as good pieces and bad pieces during the production run. This should be linked to the main consumed count of the machine. If a filler, this should be bottles into the filler.
	* Operating Time is defined as the amount of time the machine has been attempting to produce parts. (Same as above)
	* Ideal Run Rate is defined as the ideal rate that the machine can run for the product that is being run on the machine and the way the machine is configured.
	*)
	// Performance = Total Pieces / (Operating Time * Ideal Run Rate / 60)
	#OEEPerformance := (DINT_TO_REAL(#totalProdProcessed - #statTotalProdProcessed_In)) / ((#tempTimeSinceLastReset * #machineDesignSpeed / 60.0));
	IF #OEEPerformance > 1.0 THEN #OEEPerformance := 1.0; END_IF;
	IF #OEEPerformance < 0.0 THEN #OEEPerformance := 0.0; END_IF;
	
	(*  9.1.3 Quality Definition
	Quality is defined as the total number of good pieces divided by the total number of pieces on which the machine operated.
	* Quality = Good Pieces / Total Pieces
	* Good Pieces is defined as only good pieces processed during the production run. So this is the main production processed count of the machine. If a filler, this should be bottles out of the filler.
	* Total Pieces includes good pieces and bad pieces during the production run. This should be linked to the main consumed count of the machine. 
	   If a filler, this should be bottles into the filler. This should be the same count as used in the performance definition.
	*)
	// Quality = Good Piece / Total Piece
	#tempTotalProducts     :=  DINT_TO_REAL(#totalProdProcessed-#statTotalProdProcessed_In);
	#tempDefectiveProducts :=  DINT_TO_REAL(#totalDefectiveProd-#statTotalDefectiveProd_In);
	
	// Prevent divide by zero errors by checking if Total Products <> 0.0
	IF (#totalProdProcessed - #statTotalProdProcessed_In) = 0 THEN 
	    #tempTotalProducts := 0.0001;
	END_IF;
	
	// Make sure that defective products < total products
	IF #tempDefectiveProducts > #tempTotalProducts THEN
	    #tempDefectiveProducts := 0.0;
	END_IF;
	
	#OEEQuality            := (#tempTotalProducts - #tempDefectiveProducts) / #tempTotalProducts;
	
	IF #OEEQuality  > 1.0 THEN #OEEQuality  := 1.0; END_IF;
	IF #OEEQuality  < 0.0 THEN #OEEQuality  := 0.0; END_IF;
	IF #tempTotalProducts = 0 THEN
	    #OEEQuality := 0.0;
	END_IF;
	
	
	#OEERealTimeValue := #OEEAvailability * #OEEPerformance * #OEEQuality;
	
	//  -------------- END OF LOGIC -------------------------
	ENO := TRUE;   // Set the ENO output
	 
	
END_FUNCTION_BLOCK

FUNCTION_BLOCK "UN_07_RecipeControl"   // FB31627, LAD
TITLE = UN_07_RecipeControl
{ S7_Optimized_Access := 'TRUE' }
AUTHOR : tech.team.motioncontrol@siemens.com
FAMILY : CPG
VERSION : 1.0
// Support: tech.team.motioncontrol@siemens.com
// stored: AutoNumber true, IsIECCheckEnabled false, IsRetainMemResEnabled false, MemoryReserve 100, SetENOAutomatically false, UDAEnableTagReadback false
   VAR
      instRecipeControl { ExternalAccessible := 'False'; ExternalVisible := 'False'; ExternalWritable := 'False'; S7_SetPoint := 'True'} : "CPG_RecipeControl";
      instRecipeManager { ExternalAccessible := 'False'; ExternalVisible := 'False'; ExternalWritable := 'False'; S7_SetPoint := 'True'} : "CPG_RecipeHMIManager";
      ONS_RecipeChange { ExternalAccessible := 'False'; ExternalVisible := 'False'; ExternalWritable := 'False'} : Bool;
      ONS_SaveAsChange { ExternalAccessible := 'False'; ExternalVisible := 'False'; ExternalWritable := 'False'} : Bool;
      ONS_DeleteChange { ExternalAccessible := 'False'; ExternalVisible := 'False'; ExternalWritable := 'False'} : Bool;
      ONS_CopyChange { ExternalAccessible := 'False'; ExternalVisible := 'False'; ExternalWritable := 'False'} : Bool;
   END_VAR
   VAR_TEMP
      tempEnablechange : Bool;
      tempRecipenewname : String[60];
      tempErrorID : Word;
      tempError : Word;
      tempSeconds : Time;
   END_VAR
   VAR CONSTANT
      ERR_CHANGE : Word := 16#8001;
      ERR_SAVE : Word := 16#8002;
      ERR_COPY : Word := 16#8004;
      ERR_DELETE : Word := 16#8008;
   END_VAR
   VAR_TEMP   // added for the SCL form of the ladder/FBD networks
      _w1 : Bool;
      _w2 : Bool;
   END_VAR
BEGIN

REGION Network 1: Determine if recipe change is permitted based on machine state
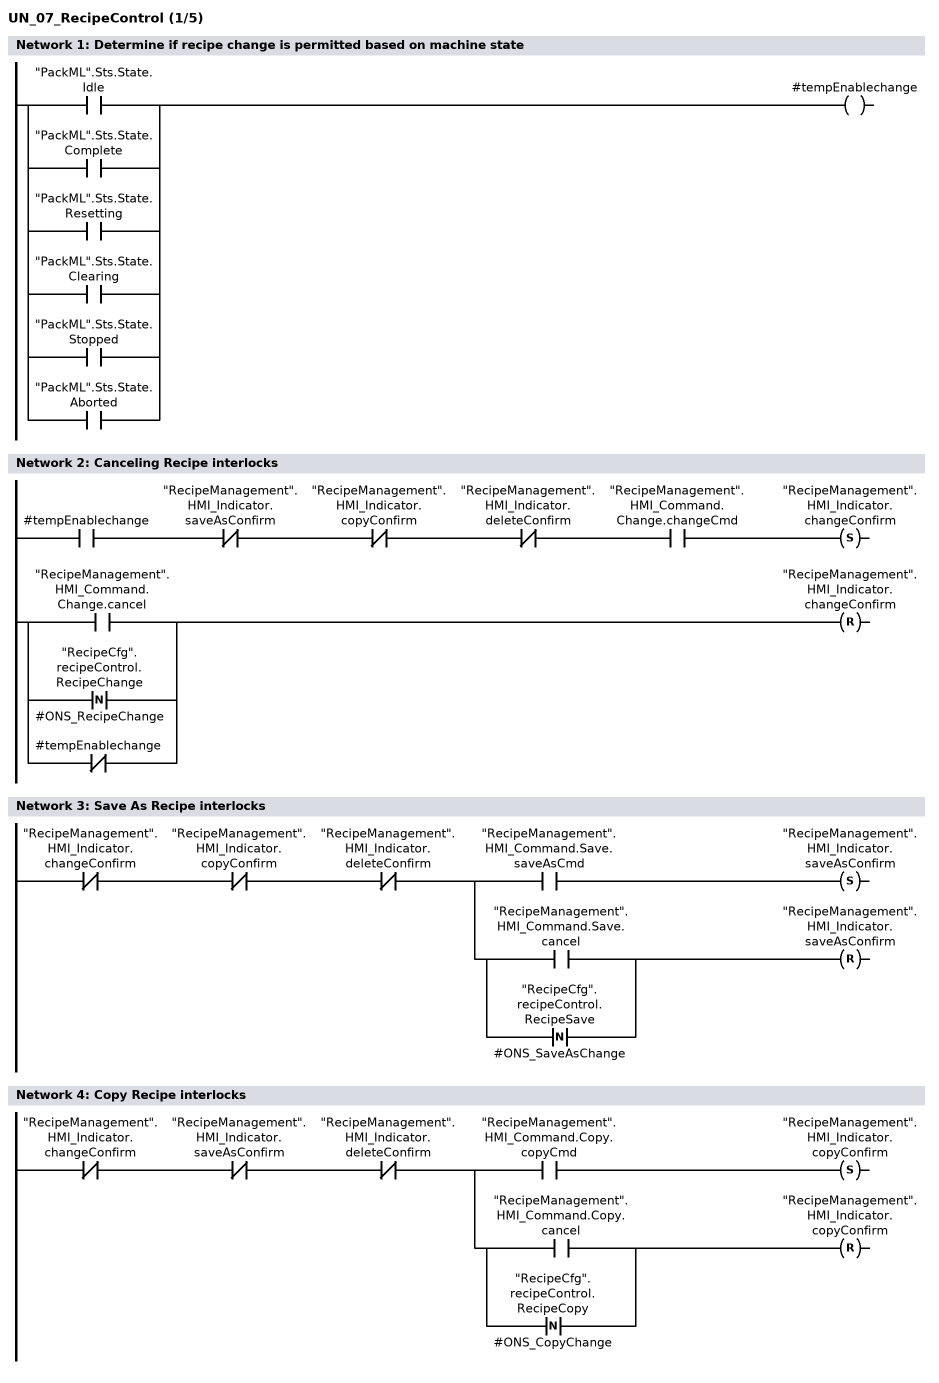
   RUNG wire#powerrail
      Contact( "PackML".Sts.State.Idle )
      wire#w1
      Coil( #tempEnablechange )
   END_RUNG
   RUNG wire#powerrail
      Contact( "PackML".Sts.State.Complete )
   END_RUNG wire#w1
   RUNG wire#powerrail
      Contact( "PackML".Sts.State.Resetting )
   END_RUNG wire#w1
   RUNG wire#powerrail
      Contact( "PackML".Sts.State.Clearing )
   END_RUNG wire#w1
   RUNG wire#powerrail
      Contact( "PackML".Sts.State.Stopped )
   END_RUNG wire#w1
   RUNG wire#powerrail
      Contact( "PackML".Sts.State.Aborted )
   END_RUNG wire#w1
   // the same network as SCL:
   #tempEnablechange := "PackML".Sts.State.Idle OR "PackML".Sts.State.Complete OR "PackML".Sts.State.Resetting OR "PackML".Sts.State.Clearing OR "PackML".Sts.State.Stopped OR "PackML".Sts.State.Aborted;
END_REGION

REGION Network 2: Canceling Recipe interlocks
   RUNG wire#powerrail
      Contact( #tempEnablechange )
      I_Contact( "RecipeManagement".HMI_Indicator.saveAsConfirm )
      I_Contact( "RecipeManagement".HMI_Indicator.copyConfirm )
      I_Contact( "RecipeManagement".HMI_Indicator.deleteConfirm )
      Contact( "RecipeManagement".HMI_Command.Change.changeCmd )
      S_Coil( "RecipeManagement".HMI_Indicator.changeConfirm )
   END_RUNG
   RUNG wire#powerrail
      Contact( "RecipeManagement".HMI_Command.Change.cancel )
      wire#w1
      R_Coil( "RecipeManagement".HMI_Indicator.changeConfirm )
   END_RUNG
   RUNG wire#powerrail
      N_Contact(operand := "RecipeCfg".recipeControl.RecipeChange, bit := #ONS_RecipeChange)
   END_RUNG wire#w1
   RUNG wire#powerrail
      I_Contact( #tempEnablechange )
   END_RUNG wire#w1
   // the same network as SCL:
   IF #tempEnablechange AND NOT "RecipeManagement".HMI_Indicator.saveAsConfirm AND NOT "RecipeManagement".HMI_Indicator.copyConfirm AND NOT "RecipeManagement".HMI_Indicator.deleteConfirm AND "RecipeManagement".HMI_Command.Change.changeCmd THEN
       "RecipeManagement".HMI_Indicator.changeConfirm := TRUE;
   END_IF;
   #_w1 := NOT "RecipeCfg".recipeControl.RecipeChange AND #ONS_RecipeChange;   // falling edge of "RecipeCfg".recipeControl.RecipeChange
   #ONS_RecipeChange := "RecipeCfg".recipeControl.RecipeChange;
   IF "RecipeManagement".HMI_Command.Change.cancel OR #_w1 OR NOT #tempEnablechange THEN
       "RecipeManagement".HMI_Indicator.changeConfirm := FALSE;
   END_IF;
END_REGION

REGION Network 3: Save As Recipe interlocks
   RUNG wire#powerrail
      I_Contact( "RecipeManagement".HMI_Indicator.changeConfirm )
      I_Contact( "RecipeManagement".HMI_Indicator.copyConfirm )
      I_Contact( "RecipeManagement".HMI_Indicator.deleteConfirm )
      wire#w1
      Contact( "RecipeManagement".HMI_Command.Save.saveAsCmd )
      S_Coil( "RecipeManagement".HMI_Indicator.saveAsConfirm )
   END_RUNG
   RUNG wire#w1
      Contact( "RecipeManagement".HMI_Command.Save.cancel )
      wire#w2
      R_Coil( "RecipeManagement".HMI_Indicator.saveAsConfirm )
   END_RUNG
   RUNG wire#w1
      N_Contact(operand := "RecipeCfg".recipeControl.RecipeSave, bit := #ONS_SaveAsChange)
   END_RUNG wire#w2
   // the same network as SCL:
   #_w1 := NOT "RecipeManagement".HMI_Indicator.changeConfirm AND NOT "RecipeManagement".HMI_Indicator.copyConfirm AND NOT "RecipeManagement".HMI_Indicator.deleteConfirm;
   IF #_w1 AND "RecipeManagement".HMI_Command.Save.saveAsCmd THEN
       "RecipeManagement".HMI_Indicator.saveAsConfirm := TRUE;
   END_IF;
   #_w2 := #_w1 AND NOT "RecipeCfg".recipeControl.RecipeSave AND #ONS_SaveAsChange;   // falling edge of "RecipeCfg".recipeControl.RecipeSave
   #ONS_SaveAsChange := "RecipeCfg".recipeControl.RecipeSave;
   IF (#_w1 AND "RecipeManagement".HMI_Command.Save.cancel) OR #_w2 THEN
       "RecipeManagement".HMI_Indicator.saveAsConfirm := FALSE;
   END_IF;
END_REGION

REGION Network 4: Copy Recipe interlocks
   RUNG wire#powerrail
      I_Contact( "RecipeManagement".HMI_Indicator.changeConfirm )
      I_Contact( "RecipeManagement".HMI_Indicator.saveAsConfirm )
      I_Contact( "RecipeManagement".HMI_Indicator.deleteConfirm )
      wire#w1
      Contact( "RecipeManagement".HMI_Command.Copy.copyCmd )
      S_Coil( "RecipeManagement".HMI_Indicator.copyConfirm )
   END_RUNG
   RUNG wire#w1
      Contact( "RecipeManagement".HMI_Command.Copy.cancel )
      wire#w2
      R_Coil( "RecipeManagement".HMI_Indicator.copyConfirm )
   END_RUNG
   RUNG wire#w1
      N_Contact(operand := "RecipeCfg".recipeControl.RecipeCopy, bit := #ONS_CopyChange)
   END_RUNG wire#w2
   // the same network as SCL:
   #_w1 := NOT "RecipeManagement".HMI_Indicator.changeConfirm AND NOT "RecipeManagement".HMI_Indicator.saveAsConfirm AND NOT "RecipeManagement".HMI_Indicator.deleteConfirm;
   IF #_w1 AND "RecipeManagement".HMI_Command.Copy.copyCmd THEN
       "RecipeManagement".HMI_Indicator.copyConfirm := TRUE;
   END_IF;
   #_w2 := #_w1 AND NOT "RecipeCfg".recipeControl.RecipeCopy AND #ONS_CopyChange;   // falling edge of "RecipeCfg".recipeControl.RecipeCopy
   #ONS_CopyChange := "RecipeCfg".recipeControl.RecipeCopy;
   IF (#_w1 AND "RecipeManagement".HMI_Command.Copy.cancel) OR #_w2 THEN
       "RecipeManagement".HMI_Indicator.copyConfirm := FALSE;
   END_IF;
END_REGION

REGION Network 5: Delete Recipe interlocks
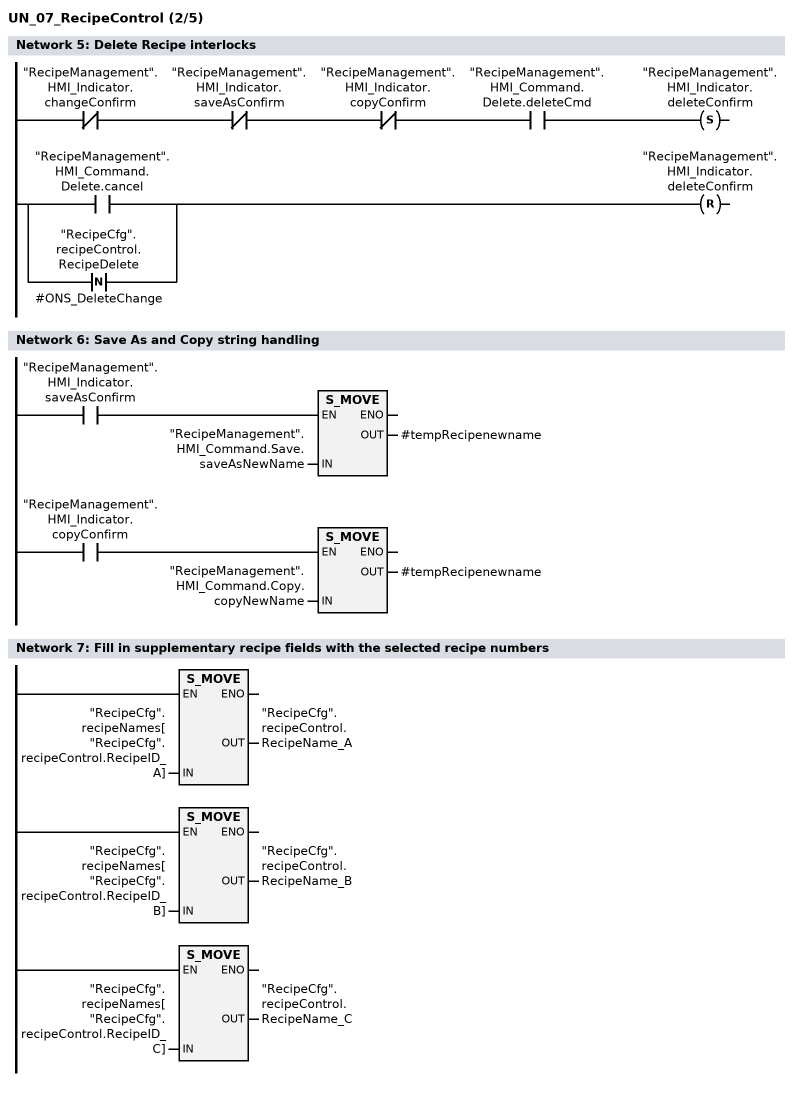
   RUNG wire#powerrail
      I_Contact( "RecipeManagement".HMI_Indicator.changeConfirm )
      I_Contact( "RecipeManagement".HMI_Indicator.saveAsConfirm )
      I_Contact( "RecipeManagement".HMI_Indicator.copyConfirm )
      Contact( "RecipeManagement".HMI_Command.Delete.deleteCmd )
      S_Coil( "RecipeManagement".HMI_Indicator.deleteConfirm )
   END_RUNG
   RUNG wire#powerrail
      Contact( "RecipeManagement".HMI_Command.Delete.cancel )
      wire#w1
      R_Coil( "RecipeManagement".HMI_Indicator.deleteConfirm )
   END_RUNG
   RUNG wire#powerrail
      N_Contact(operand := "RecipeCfg".recipeControl.RecipeDelete, bit := #ONS_DeleteChange)
   END_RUNG wire#w1
   // the same network as SCL:
   IF NOT "RecipeManagement".HMI_Indicator.changeConfirm AND NOT "RecipeManagement".HMI_Indicator.saveAsConfirm AND NOT "RecipeManagement".HMI_Indicator.copyConfirm AND "RecipeManagement".HMI_Command.Delete.deleteCmd THEN
       "RecipeManagement".HMI_Indicator.deleteConfirm := TRUE;
   END_IF;
   #_w1 := NOT "RecipeCfg".recipeControl.RecipeDelete AND #ONS_DeleteChange;   // falling edge of "RecipeCfg".recipeControl.RecipeDelete
   #ONS_DeleteChange := "RecipeCfg".recipeControl.RecipeDelete;
   IF "RecipeManagement".HMI_Command.Delete.cancel OR #_w1 THEN
       "RecipeManagement".HMI_Indicator.deleteConfirm := FALSE;
   END_IF;
END_REGION

REGION Network 6: Save As and Copy string handling
   RUNG wire#powerrail
      Contact( "RecipeManagement".HMI_Indicator.saveAsConfirm )
      S_Move(in := "RecipeManagement".HMI_Command.Save.saveAsNewName, out => #tempRecipenewname)
   END_RUNG
   RUNG wire#powerrail
      Contact( "RecipeManagement".HMI_Indicator.copyConfirm )
      S_Move(in := "RecipeManagement".HMI_Command.Copy.copyNewName, out => #tempRecipenewname)
   END_RUNG
   // the same network as SCL:
   IF "RecipeManagement".HMI_Indicator.saveAsConfirm THEN
       #tempRecipenewname := "RecipeManagement".HMI_Command.Save.saveAsNewName;
   END_IF;
   IF "RecipeManagement".HMI_Indicator.copyConfirm THEN
       #tempRecipenewname := "RecipeManagement".HMI_Command.Copy.copyNewName;
   END_IF;
END_REGION

REGION Network 7: Fill in supplementary recipe fields with the selected recipe numbers
   RUNG wire#powerrail
      S_Move(in := "RecipeCfg".recipeNames["RecipeCfg".recipeControl.RecipeID_A], out => "RecipeCfg".recipeControl.RecipeName_A)
   END_RUNG
   RUNG wire#powerrail
      S_Move(in := "RecipeCfg".recipeNames["RecipeCfg".recipeControl.RecipeID_B], out => "RecipeCfg".recipeControl.RecipeName_B)
   END_RUNG
   RUNG wire#powerrail
      S_Move(in := "RecipeCfg".recipeNames["RecipeCfg".recipeControl.RecipeID_C], out => "RecipeCfg".recipeControl.RecipeName_C)
   END_RUNG
   // the same network as SCL:
   "RecipeCfg".recipeControl.RecipeName_A := "RecipeCfg".recipeNames["RecipeCfg".recipeControl.RecipeID_A];
   "RecipeCfg".recipeControl.RecipeName_B := "RecipeCfg".recipeNames["RecipeCfg".recipeControl.RecipeID_B];
   "RecipeCfg".recipeControl.RecipeName_C := "RecipeCfg".recipeNames["RecipeCfg".recipeControl.RecipeID_C];
END_REGION

REGION Network 8: Call Recipe Control
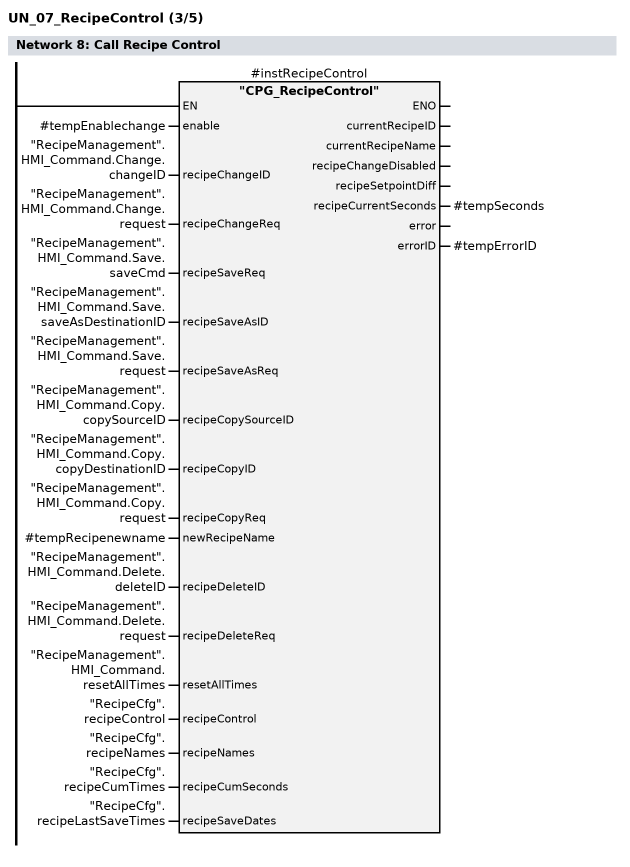
   RUNG wire#powerrail
      #instRecipeControl(enable := #tempEnablechange, recipeChangeID := "RecipeManagement".HMI_Command.Change.changeID, recipeChangeReq := "RecipeManagement".HMI_Command.Change.request, recipeSaveReq := "RecipeManagement".HMI_Command.Save.saveCmd, recipeSaveAsID := "RecipeManagement".HMI_Command.Save.saveAsDestinationID, recipeSaveAsReq := "RecipeManagement".HMI_Command.Save.request, recipeCopySourceID := "RecipeManagement".HMI_Command.Copy.copySourceID, recipeCopyID := "RecipeManagement".HMI_Command.Copy.copyDestinationID, recipeCopyReq := "RecipeManagement".HMI_Command.Copy.request, newRecipeName := #tempRecipenewname, recipeDeleteID := "RecipeManagement".HMI_Command.Delete.deleteID, recipeDeleteReq := "RecipeManagement".HMI_Command.Delete.request, resetAllTimes := "RecipeManagement".HMI_Command.resetAllTimes, recipeControl := "RecipeCfg".recipeControl, recipeNames := "RecipeCfg".recipeNames, recipeCumSeconds := "RecipeCfg".recipeCumTimes, recipeSaveDates := "RecipeCfg".recipeLastSaveTimes, currentRecipeID =>, currentRecipeName =>, recipeChangeDisabled =>, recipeSetpointDiff =>, recipeCurrentSeconds => #tempSeconds, error =>, errorID => #tempErrorID)
   END_RUNG
   // the same network as SCL:
   #instRecipeControl(enable := #tempEnablechange,   // "CPG_RecipeControl"
                      recipeChangeID := "RecipeManagement".HMI_Command.Change.changeID,
                      recipeChangeReq := "RecipeManagement".HMI_Command.Change.request,
                      recipeSaveReq := "RecipeManagement".HMI_Command.Save.saveCmd,
                      recipeSaveAsID := "RecipeManagement".HMI_Command.Save.saveAsDestinationID,
                      recipeSaveAsReq := "RecipeManagement".HMI_Command.Save.request,
                      recipeCopySourceID := "RecipeManagement".HMI_Command.Copy.copySourceID,
                      recipeCopyID := "RecipeManagement".HMI_Command.Copy.copyDestinationID,
                      recipeCopyReq := "RecipeManagement".HMI_Command.Copy.request,
                      newRecipeName := #tempRecipenewname,
                      recipeDeleteID := "RecipeManagement".HMI_Command.Delete.deleteID,
                      recipeDeleteReq := "RecipeManagement".HMI_Command.Delete.request,
                      resetAllTimes := "RecipeManagement".HMI_Command.resetAllTimes,
                      recipeControl := "RecipeCfg".recipeControl,
                      recipeNames := "RecipeCfg".recipeNames,
                      recipeCumSeconds := "RecipeCfg".recipeCumTimes,
                      recipeSaveDates := "RecipeCfg".recipeLastSaveTimes,
                      recipeCurrentSeconds => #tempSeconds,
                      errorID => #tempErrorID);
END_REGION

